# B&R Automation Studio project PLC code - cp (part 19)

#### InputsMecano.st - PhysicalInputs
```iecst
ACTION InputsMecano:

	//////////
	//PRINTER
	//////////

	// Machine controlled by line. Always with consent
	gMachine.In.xConsentL1Ok := TRUE;
	gMachine.In.xConsentL2Ok := TRUE;

	//Digital Inputs
	gMachine.In.Buttons.xStart := X20DIF371_101.DInput[1];
	gMachine.In.Buttons.xStop := NOT X20DIF371_101.DInput[2];
	gMachine.In.Buttons.xAuto := X20DIF371_101.DInput[3];
	gMachine.In.Buttons.xZero := NOT X20DIF371_101.DInput[4];
	gMachine.In.Buttons.xManual := X20DIF371_101.DInput[5];
	gMachine.In.Buttons.xReset := X20DIF371_101.DInput[6];
	//Back Safety Key unlock - PRINTER := X20DIF371_101.DInput[7];
	gBlockInputs[1].xReferenceDI := X20DIF371_101.DInput[8];
	gJamInputs[1].xJamLowCrash := X20DIF371_101.DInput[9];
	gJamInputs[2].xJamLowCrash := X20DIF371_101.DInput[10];
	gJamInputs[3].xJamLowCrash := X20DIF371_101.DInput[11];
	gJamInputs[1].xJamTestOk := X20DIF371_101.DInput[13];
	gJamInputs[2].xJamTestOk := X20DIF371_101.DInput[14];
	gJamInputs[3].xJamTestOk := X20DIF371_101.DInput[15];

	gBlockInputs[1].xPrintHeadPSU[1] := X20DIF371_102.DInput[1];
	gBlockInputs[1].xPrintHeadPSU[2] := X20DIF371_102.DInput[2];
	gBlockInputs[1].xPrintHeadPSU[3] := X20DIF371_102.DInput[3];
	gBlockInputs[1].xHeaterDcOkPsu[1] := gBlockInputs[1].xHeaterAcOkPsu[1] := X20DIF371_102.DInput[4];
	gInksInputs[3].xPrintHeadsPsuOK := X20DIF371_102.DInput[5];
	gInksInputs[4].xPrintHeadsPsuOK := X20DIF371_102.DInput[6];
	gInksInputs[5].xPrintHeadsPsuOK := X20DIF371_102.DInput[7];
	gInksInputs[6].xPrintHeadsPsuOK := X20DIF371_102.DInput[8];
	gInksInputs[7].xPrintHeadsPsuOK := X20DIF371_102.DInput[9];
	gInksInputs[8].xPrintHeadsPsuOK := X20DIF371_102.DInput[10];
	gInksInputs[9].xPrintHeadsPsuOK := X20DIF371_102.DInput[11];
	gInksInputs[10].xPrintHeadsPsuOK := X20DIF371_102.DInput[12];
	gMachine.In.x24Vdc := X20DIF371_102.DInput[13];
	gBelt.parameters.xDriveProtectionOK := X20DIF371_102.DInput[14];
	gBlockInputs[1].xDriveProtectionOK := gBlockInputs[1].xDifferentialOK := X20DIF371_102.DInput[15];
	FOR iIndexCuringLed:=1 TO MAX_LAST_CURING_LED DO
		gCuringLed[iIndexCuringLed].Signals.Inputs.xFrontDoorClosed := X20DIF371_102.DInput[16];
	END_FOR

	gMachine.In.ProductDetect.pPDSignalSensorL1	:= ADR(X20DIF371_103.DInput[1]);
	gMachine.In.ProductDetect.pPDSignalSensorL2	:= ADR(X20DIF371_103.DInput[2]);
	gPhotoCells.Inputs.Signals.pInput[1] := ADR(X20DIF371_103.DInput[3]);
	gPhotoCells.Inputs.Signals.pInput[2] := ADR(X20DIF371_103.DInput[4]);
	gPhotoCells.Inputs.Signals.pInput[3] := ADR(X20DIF371_103.DInput[5]);
	gPhotoCells.Inputs.Signals.pInput[4] := ADR(X20DIF371_103.DInput[6]);
	gPhotoCells.Inputs.Signals.pInput[5] := ADR(X20DIF371_103.DInput[7]);
	gPhotoCells.Inputs.Signals.pInput[6] := ADR(X20DIF371_103.DInput[8]);
	gPhotoCells.Inputs.Signals.xSafetyEnable := gMachine.In.xSafetyEnabled;

	gJamInputs[1].xJamCrash[1] := X20DIF371_104.DInput[1];
	gJamInputs[1].xJamCrash[2] := X20DIF371_104.DInput[2];
	gJamInputs[1].xJamCrash[3] := X20DIF371_104.DInput[3];
	gJamInputs[1].xJamCrash[4] := X20DIF371_104.DInput[4];
	gJamInputs[2].xJamCrash[1] := X20DIF371_104.DInput[5];
	gJamInputs[2].xJamCrash[2] := X20DIF371_104.DInput[6];
	gJamInputs[2].xJamCrash[3] := X20DIF371_104.DInput[7];
	gJamInputs[2].xJamCrash[4] := X20DIF371_104.DInput[8];
	gJamInputs[3].xJamCrash[1] := X20DIF371_104.DInput[9];
	gJamInputs[3].xJamCrash[2] := X20DIF371_104.DInput[10];

	gInksInputs[3].xKlixonTriggered := X20DIF371_105.DInput[1];
	gInksInputs[4].xKlixonTriggered := X20DIF371_105.DInput[2];
	gInksInputs[5].xKlixonTriggered := X20DIF371_105.DInput[3];
	gInksInputs[6].xKlixonTriggered := X20DIF371_105.DInput[4];
	gInksInputs[7].xKlixonTriggered := X20DIF371_105.DInput[5];
	gInksInputs[8].xKlixonTriggered := X20DIF371_105.DInput[6];
	gInksInputs[9].xKlixonTriggered := X20DIF371_105.DInput[7];
	gInksInputs[10].xKlixonTriggered := X20DIF371_105.DInput[8];

	gInksInputs[3].xOverpressure  := NOT X20DIF371_105.DInput[9];
	gInksInputs[4].xOverpressure  := NOT X20DIF371_105.DInput[10];
	gInksInputs[5].xOverpressure  := NOT X20DIF371_105.DInput[11];
	gInksInputs[6].xOverpressure  := NOT X20DIF371_105.DInput[12];
	gInksInputs[7].xOverpressure  := NOT X20DIF371_105.DInput[13];
	gInksInputs[8].xOverpressure  := NOT X20DIF371_105.DInput[14];
	gInksInputs[9].xOverpressure  := NOT X20DIF371_105.DInput[15];
	gInksInputs[10].xOverpressure  := NOT X20DIF371_105.DInput[16];

	gInksInputs[3].xConnected := X20DIF371_106.DInput[1];
	gInksInputs[4].xConnected := X20DIF371_106.DInput[2];
	gInksInputs[5].xConnected := X20DIF371_106.DInput[3];
	gInksInputs[6].xConnected := X20DIF371_106.DInput[4];
	gInksInputs[7].xConnected := X20DIF371_106.DInput[5];
	gInksInputs[8].xConnected := X20DIF371_106.DInput[6];
	gInksInputs[9].xConnected := X20DIF371_106.DInput[7];
	gInksInputs[10].xConnected := X20DIF371_106.DInput[8];

	//Analog inputs
	gTransVacuum[1].Inputs.iPressureRaw := X20AI8321_111.AInput[1];
	gTransVacuum[1].Inputs.xPressureSensorError := StatusAnalogInputBroken( X20AI8321_111.ModuleOk, X20AI8321_111.Status01, X20AI8321_111.Status02, 1);
	gTransVacuum[2].Inputs.iPressureRaw := X20AI8321_111.AInput[2];
	gTransVacuum[2].Inputs.xPressureSensorError := StatusAnalogInputBroken( X20AI8321_111.ModuleOk, X20AI8321_111.Status01, X20AI8321_111.Status02, 2);

	gInksInputs[3].iVacuum1Raw := X20AI8321_112.AInput[1];
	gInksInputs[3].xVacuum1SensorError 	:= StatusAnalogInputBroken( X20AI8321_112.ModuleOk, X20AI8321_112.Status01, X20AI8321_112.Status02, 1);
	gInksInputs[3].iVacuum2Raw := X20AI8321_112.AInput[2];
	gInksInputs[3].xVacuum2SensorError 	:= StatusAnalogInputBroken( X20AI8321_112.ModuleOk, X20AI8321_112.Status01, X20AI8321_112.Status02, 2);
	gInksInputs[4].iVacuum1Raw := X20AI8321_112.AInput[3];
	gInksInputs[4].xVacuum1SensorError 	:= StatusAnalogInputBroken( X20AI8321_112.ModuleOk, X20AI8321_112.Status01, X20AI8321_112.Status02, 3);
	gInksInputs[4].iVacuum2Raw := X20AI8321_112.AInput[4];
	gInksInputs[4].xVacuum2SensorError 	:= StatusAnalogInputBroken( X20AI8321_112.ModuleOk, X20AI8321_112.Status01, X20AI8321_112.Status02, 4);
	gInksInputs[5].iVacuum1Raw := X20AI8321_112.AInput[5];
	gInksInputs[5].xVacuum1SensorError 	:= StatusAnalogInputBroken( X20AI8321_112.ModuleOk, X20AI8321_112.Status01, X20AI8321_112.Status02, 5);
	gInksInputs[5].iVacuum2Raw := X20AI8321_112.AInput[6];
	gInksInputs[5].xVacuum2SensorError 	:= StatusAnalogInputBroken( X20AI8321_112.ModuleOk, X20AI8321_112.Status01, X20AI8321_112.Status02, 6);
	gInksInputs[6].iVacuum1Raw := X20AI8321_112.AInput[7];
	gInksInputs[6].xVacuum1SensorError 	:= StatusAnalogInputBroken( X20AI8321_112.ModuleOk, X20AI8321_112.Status01, X20AI8321_112.Status02, 7);
	gInksInputs[6].iVacuum2Raw := X20AI8321_112.AInput[8];
	gInksInputs[6].xVacuum2SensorError 	:= StatusAnalogInputBroken( X20AI8321_112.ModuleOk, X20AI8321_112.Status01, X20AI8321_112.Status02, 8);

	gInksInputs[7].iVacuum1Raw := X20AI8321_113.AInput[1];
	gInksInputs[7].xVacuum1SensorError 	:= StatusAnalogInputBroken( X20AI8321_113.ModuleOk, X20AI8321_113.Status01, X20AI8321_113.Status02, 1);
	gInksInputs[7].iVacuum2Raw := X20AI8321_113.AInput[2];
	gInksInputs[7].xVacuum2SensorError 	:= StatusAnalogInputBroken( X20AI8321_113.ModuleOk, X20AI8321_113.Status01, X20AI8321_113.Status02, 2);
	gInksInputs[8].iVacuum1Raw := X20AI8321_113.AInput[3];
	gInksInputs[8].xVacuum1SensorError 	:= StatusAnalogInputBroken( X20AI8321_113.ModuleOk, X20AI8321_113.Status01, X20AI8321_113.Status02, 3);
	gInksInputs[8].iVacuum2Raw := X20AI8321_113.AInput[4];
	gInksInputs[8].xVacuum2SensorError 	:= StatusAnalogInputBroken( X20AI8321_113.ModuleOk, X20AI8321_113.Status01, X20AI8321_113.Status02, 4);
	gInksInputs[9].iVacuum1Raw := X20AI8321_113.AInput[5];
	gInksInputs[9].xVacuum1SensorError 	:= StatusAnalogInputBroken( X20AI8321_113.ModuleOk, X20AI8321_113.Status01, X20AI8321_113.Status02, 5);
	gInksInputs[9].iVacuum2Raw := X20AI8321_113.AInput[6];
	gInksInputs[9].xVacuum2SensorError 	:= StatusAnalogInputBroken( X20AI8321_113.ModuleOk, X20AI8321_113.Status01, X20AI8321_113.Status02, 6);
	gInksInputs[10].iVacuum1Raw := X20AI8321_113.AInput[7];
	gInksInputs[10].xVacuum1SensorError 	:= StatusAnalogInputBroken( X20AI8321_113.ModuleOk, X20AI8321_113.Status01, X20AI8321_113.Status02, 7);
	gInksInputs[10].iVacuum2Raw := X20AI8321_113.AInput[8];
	gInksInputs[10].xVacuum2SensorError 	:= StatusAnalogInputBroken( X20AI8321_113.ModuleOk, X20AI8321_113.Status01, X20AI8321_113.Status02, 8);

	gInksInputs[3].iInTankLevel := X20AI8321_114.AInput[1];
	gInksInputs[3].xInkLevelTankSensorError := StatusAnalogInputBroken( X20AI8321_114.ModuleOk, X20AI8321_114.Status01, X20AI8321_114.Status02, 1);
	gInksInputs[4].iInTankLevel := X20AI8321_114.AInput[2];
	gInksInputs[4].xInkLevelTankSensorError := StatusAnalogInputBroken( X20AI8321_114.ModuleOk, X20AI8321_114.Status01, X20AI8321_114.Status02, 2);
	gInksInputs[5].iInTankLevel := X20AI8321_114.AInput[3];
	gInksInputs[5].xInkLevelTankSensorError := StatusAnalogInputBroken( X20AI8321_114.ModuleOk, X20AI8321_114.Status01, X20AI8321_114.Status02, 3);
	gInksInputs[6].iInTankLevel := X20AI8321_114.AInput[4];
	gInksInputs[6].xInkLevelTankSensorError := StatusAnalogInputBroken( X20AI8321_114.ModuleOk, X20AI8321_114.Status01, X20AI8321_114.Status02, 4);
	gInksInputs[7].iInTankLevel := X20AI8321_114.AInput[5];
	gInksInputs[7].xInkLevelTankSensorError := StatusAnalogInputBroken( X20AI8321_114.ModuleOk, X20AI8321_114.Status01, X20AI8321_114.Status02, 5);
	gInksInputs[8].iInTankLevel := X20AI8321_114.AInput[6];
	gInksInputs[8].xInkLevelTankSensorError := StatusAnalogInputBroken( X20AI8321_114.ModuleOk, X20AI8321_114.Status01, X20AI8321_114.Status02, 6);
	gInksInputs[9].iInTankLevel := X20AI8321_114.AInput[7];
	gInksInputs[9].xInkLevelTankSensorError := StatusAnalogInputBroken( X20AI8321_114.ModuleOk, X20AI8321_114.Status01, X20AI8321_114.Status02, 7);
	gInksInputs[10].iInTankLevel := X20AI8321_114.AInput[8];
	gInksInputs[10].xInkLevelTankSensorError := StatusAnalogInputBroken( X20AI8321_114.ModuleOk, X20AI8321_114.Status01, X20AI8321_114.Status02, 8);

	//PT100
	gBlockInputs[1].xModuleTemp01Ok	:= X20AT4222_120.ModuleOk;
	gInksInputs[3].iTemperatureRaw := X20AT4222_120.TempInput[1];
	gInksInputs[3].xTempSensorError	:= StatusTemperatureInput(X20AT4222_120.Status01, 1);
	gInksInputs[4].iTemperatureRaw := X20AT4222_120.TempInput[2];
	gInksInputs[4].xTempSensorError	:= StatusTemperatureInput(X20AT4222_120.Status01, 2);
	gInksInputs[5].iTemperatureRaw := X20AT4222_120.TempInput[3];
	gInksInputs[5].xTempSensorError	:= StatusTemperatureInput(X20AT4222_120.Status01, 3);
	gInksInputs[6].iTemperatureRaw := X20AT4222_120.TempInput[4];
	gInksInputs[6].xTempSensorError	:= StatusTemperatureInput(X20AT4222_120.Status01, 4);

	gBlockInputs[1].xModuleTemp02Ok	:= X20AT4222_121.ModuleOk;
	gInksInputs[7].iTemperatureRaw := X20AT4222_121.TempInput[1];
	gInksInputs[7].xTempSensorError	:= StatusTemperatureInput(X20AT4222_121.Status01, 1);
	gInksInputs[8].iTemperatureRaw := X20AT4222_121.TempInput[2];
	gInksInputs[8].xTempSensorError	:= StatusTemperatureInput(X20AT4222_121.Status01, 2);
	gInksInputs[9].iTemperatureRaw := X20AT4222_121.TempInput[3];
	gInksInputs[9].xTempSensorError	:= StatusTemperatureInput(X20AT4222_121.Status01, 3);
	gInksInputs[10].iTemperatureRaw := X20AT4222_121.TempInput[4];
	gInksInputs[10].xTempSensorError	:= StatusTemperatureInput(X20AT4222_121.Status01, 4);

	// SI UNIT BK1
	gBlockInputs[1].xSiUnitModuleOk		:= SiUnitPwrLnkBK1.ModuleOk;
	gMachine.In.xAirSupply				:= SiUnitPwrLnkBK1.Input01_16.0;
	gBlockInputs[1].xAirVenturiOK		:= SiUnitPwrLnkBK1.Input01_16.1;
	gBlockInputs[1].xTrayOut			:= SiUnitPwrLnkBK1.Input01_16.2;
	gBlockInputs[1].xIclaSensor			:= SiUnitPwrLnkBK1.Input01_16.3;
	gTransVacuum[1].Inputs.xVaccAirFlow	:= gTransVacuum[2].Inputs.xVaccAirFlow := SiUnitPwrLnkBK1.Input01_16.4; //No estamos haciendo nada con esto en el package de TransVacuum!
	gTransVacuum[1].Inputs.xJointSystemPressure:= gTransVacuum[2].Inputs.xJointSystemPressure := SiUnitPwrLnkBK1.Input01_16.5;
	gMachine.In.CleanBelt.xLowPosition 	:= SiUnitPwrLnkBK1.Input01_16.6;
	gMachine.In.CleanBelt.xHighPosition := SiUnitPwrLnkBK1.Input01_16.7;
	gBlockInputs[1].xBarsIn := TRUE;
	gTransVacuum[1].Inputs.xSafetyEnable := gTransVacuum[2].Inputs.xSafetyEnable := gMachine.In.xSafetyEnabled;

	//Signals Forced by Configuration
	gBlockInputs[1].Safety.xFrontEStopOK := gSafetyController.Inputs.xPrinterFrontsideEstop;
	gBlockInputs[1].Safety.xRearEStopOK := gSafetyController.Inputs.xPrinterBacksideEstop;

	gBlockInputs[1].Safety.xFrontSafetyOK	:= gSafetyController.Inputs.xPrinterFrontsideEstop AND gSafetyController.Inputs.xPrinterLightCurtain;
	gBlockInputs[1].Safety.xRearSafetyOK	:= gSafetyController.Inputs.xPrinterBacksideEstop AND gSafetyController.Inputs.xPrinterDoorLock;
	gBlockInputs[1].Safety.xSafetyOK 		:= gMachine.In.xSafetyEnabled;

	//There are no specific enables for light curtains. So we mapp PrinterLightCurtain status to these inputs to acknowledge that curtain is crossed
	gBlockInputs[1].Safety.xCurtainEnable01 := gBlockInputs[1].Safety.xCurtainEnable02 := gSafetyController.Inputs.xPrinterLightCurtain;

	//Signals Forced by Configuration
	FOR iIndexVac := 1 TO MAX_LAST_TRANS_VACUUM DO gTransVacuum[iIndexVac].Inputs.xBlowersAnyCB := FALSE; END_FOR

	///////////////////////////
	//UV Curing leds related

	//Digital inputs
	gCuringLed[iIndexColorCuringLedBar].Lamp[1].Inputs.ThermalFault	:= NOT X20DIF371_151.DInput[1];
	gCuringLed[iIndexColorCuringLedBar].Lamp[1].Inputs.SLMFault		:= NOT X20DIF371_151.DInput[2];
	gCuringLed[iIndexColorCuringLedBar].Lamp[2].Inputs.ThermalFault	:= NOT X20DIF371_151.DInput[3];
	gCuringLed[iIndexColorCuringLedBar].Lamp[2].Inputs.SLMFault		:= NOT X20DIF371_151.DInput[4];
	gCuringLed[iIndexColorCuringLedBar].Lamp[3].Inputs.ThermalFault	:= NOT X20DIF371_151.DInput[5];
	gCuringLed[iIndexColorCuringLedBar].Lamp[3].Inputs.SLMFault		:= NOT X20DIF371_151.DInput[6];
	gCuringLed[iIndexColorCuringLedBar].Lamp[4].Inputs.ThermalFault	:= NOT X20DIF371_151.DInput[7];
	gCuringLed[iIndexColorCuringLedBar].Lamp[4].Inputs.SLMFault		:= NOT X20DIF371_151.DInput[8];
	gCuringLed[iIndexColorCuringLedBar].Lamp[5].Inputs.ThermalFault	:= NOT X20DIF371_151.DInput[9];
	gCuringLed[iIndexColorCuringLedBar].Lamp[5].Inputs.SLMFault		:= NOT X20DIF371_151.DInput[10];
	gCuringLed[iIndexColorCuringLedBar].Signals.Inputs.xN2HighFlow	:= NOT X20DIF371_151.DInput[13];
	gCuringLed[iIndexColorCuringLedBar].Signals.Inputs.xN2LowFlow	:= NOT X20DIF371_151.DInput[14];

	gCuringLed[iIndexWhiteCuringLedBar].Lamp[1].Inputs.ThermalFault	:= NOT X20DIF371_152.DInput[1];
	gCuringLed[iIndexWhiteCuringLedBar].Lamp[1].Inputs.SLMFault		:= NOT X20DIF371_152.DInput[2];
	gCuringLed[iIndexWhiteCuringLedBar].Lamp[2].Inputs.ThermalFault	:= NOT X20DIF371_152.DInput[3];
	gCuringLed[iIndexWhiteCuringLedBar].Lamp[2].Inputs.SLMFault		:= NOT X20DIF371_152.DInput[4];
	gCuringLed[iIndexWhiteCuringLedBar].Lamp[3].Inputs.ThermalFault	:= NOT X20DIF371_152.DInput[5];
	gCuringLed[iIndexWhiteCuringLedBar].Lamp[3].Inputs.SLMFault		:= NOT X20DIF371_152.DInput[6];
	gCuringLed[iIndexWhiteCuringLedBar].Lamp[4].Inputs.ThermalFault	:= NOT X20DIF371_152.DInput[7];
	gCuringLed[iIndexWhiteCuringLedBar].Lamp[4].Inputs.SLMFault		:= NOT X20DIF371_152.DInput[8];
	gCuringLed[iIndexWhiteCuringLedBar].Lamp[5].Inputs.ThermalFault	:= NOT X20DIF371_152.DInput[9];
	gCuringLed[iIndexWhiteCuringLedBar].Lamp[5].Inputs.SLMFault		:= NOT X20DIF371_152.DInput[10];
	gCuringLed[iIndexWhiteCuringLedBar].Signals.Inputs.xN2HighFlow	:= NOT X20DIF371_152.DInput[13];
	gCuringLed[iIndexWhiteCuringLedBar].Signals.Inputs.xN2LowFlow	:= NOT X20DIF371_152.DInput[14];

	gCuringLed[iIndexPrimerCuringLedBar].Lamp[1].Inputs.ThermalFault	:= NOT X20DIF371_153.DInput[1];
	gCuringLed[iIndexPrimerCuringLedBar].Lamp[1].Inputs.SLMFault		:= NOT X20DIF371_153.DInput[2];
	gCuringLed[iIndexPrimerCuringLedBar].Lamp[2].Inputs.ThermalFault	:= NOT X20DIF371_153.DInput[3];
	gCuringLed[iIndexPrimerCuringLedBar].Lamp[2].Inputs.SLMFault		:= NOT X20DIF371_153.DInput[4];
	gCuringLed[iIndexPrimerCuringLedBar].Lamp[3].Inputs.ThermalFault	:= NOT X20DIF371_153.DInput[5];
	gCuringLed[iIndexPrimerCuringLedBar].Lamp[3].Inputs.SLMFault		:= NOT X20DIF371_153.DInput[6];
	gCuringLed[iIndexPrimerCuringLedBar].Lamp[4].Inputs.ThermalFault	:= NOT X20DIF371_153.DInput[7];
	gCuringLed[iIndexPrimerCuringLedBar].Lamp[4].Inputs.SLMFault		:= NOT X20DIF371_153.DInput[8];
	gCuringLed[iIndexPrimerCuringLedBar].Lamp[5].Inputs.ThermalFault	:= NOT X20DIF371_153.DInput[9];
	gCuringLed[iIndexPrimerCuringLedBar].Lamp[5].Inputs.SLMFault		:= NOT X20DIF371_153.DInput[10];
	gCuringLed[iIndexPrimerCuringLedBar].Signals.Inputs.xN2HighFlow		:= NOT X20DIF371_153.DInput[13];
	gCuringLed[iIndexPrimerCuringLedBar].Signals.Inputs.xN2LowFlow		:= NOT X20DIF371_153.DInput[14];

	gMachine.In.CleanBelt.xError 						:= X20DIF371_154.DInput[1];
	gMachine.In.CleanBelt.xOpenGuide 					:= X20DIF371_154.DInput[2];
	gMachine.In.AntiStatic.xGenAlarm 					:= X20DIF371_154.DInput[3];
	gMachine.In.AntiStatic.xIonLevelAlarm				:= X20DIF371_154.DInput[4];

	//////////
	//PDC
	//////////
	//Line X20DIF371_002
	//These inputs are read in MachineConfigurator>InputsMachineModel
	//	:= Pdc_X20DIF371_002.DInput[1];
	//	:= Pdc_X20DIF371_002.DInput[2];
	//	:= Pdc_X20DIF371_002.DInput[3];
	//	:= Pdc_X20DIF371_002.DInput[4];
	//	:= Pdc_X20DIF371_002.DInput[5];
	//	:= Pdc_X20DIF371_002.DInput[6];
	gFeeder.Inputs.xNoPowered 					:= NOT Pdc_X20DIF371_002.DInput[7];
	gSarm.Inputs.xPowered						:= Pdc_X20DIF371_002.DInput[8];
	gPrimer.Inputs.xNoPowered 					:= NOT Pdc_X20DIF371_002.DInput[9];
	gLine.Inputs.xPrinterPowered				:= Pdc_X20DIF371_002.DInput[10];
	gOverVarnish.Inputs.xNoPowered  			:= NOT Pdc_X20DIF371_002.DInput[11];
	gStacker.Inputs.xNoPowered 					:= NOT Pdc_X20DIF371_002.DInput[12];
	gLine.Inputs.xOvervoltageProtectionOk 		:= NOT Pdc_X20DIF371_002.DInput[13]; //Inverse logic
	gMachine.In.xSafetyEnabled 					:= Pdc_X20DIF371_002.DInput[14];

	//Line X20DIF371_003
	gAxisInverter[1].ElecSignals.In.xBreakerOK 	:= Pdc_X20DIF371_003.DInput[1];
	gAxisInverter[2].ElecSignals.In.xBreakerOK 	:= Pdc_X20DIF371_003.DInput[2];
	gAxisInverter[3].ElecSignals.In.xBreakerOK 	:= Pdc_X20DIF371_003.DInput[3];
	gAxisInverter[4].ElecSignals.In.xBreakerOK 	:= Pdc_X20DIF371_003.DInput[4];
	gMachine.In.xHoppersSoftStarterFault	:= Pdc_X20DIF371_003.DInput[5];
	gLine.Inputs.UPSs[1].LoadOnUtility		:= Pdc_X20DIF371_003.DInput[6];
	gLine.Inputs.UPSs[1].LoadOnBattery 		:= gLine.Inputs.UPSs[1].xPowerFault := Pdc_X20DIF371_003.DInput[7];
	gLine.Inputs.UPSs[1].xLowBattery 		:= Pdc_X20DIF371_003.DInput[8];
	gLine.Inputs.UPSs[1].xByPass			:= Pdc_X20DIF371_003.DInput[9];
	gLine.Inputs.x24VdcStartSeqNoPowered	:= NOT Pdc_X20DIF371_003.DInput[10];

	//Line X20DIF371_004
	gFeeder.Inputs.xModelInput[0] 		:= Pdc_X20DIF371_004.DInput[1];
	gFeeder.Inputs.xModelInput[1] 		:= Pdc_X20DIF371_004.DInput[2];
	gFeeder.Inputs.xModelInput[2] 		:= Pdc_X20DIF371_004.DInput[3];
	gFeeder.Inputs.xOnline 				:= Pdc_X20DIF371_004.DInput[4];
	gFeeder.Inputs.xError 				:= Pdc_X20DIF371_004.DInput[5];
	gFeeder.Inputs.xFeeding 			:= Pdc_X20DIF371_004.DInput[6];
	gFeeder.Inputs.xMultiPick 			:= Pdc_X20DIF371_004.DInput[7];
	gFeeder.Inputs.xTrayEmpty 			:= Pdc_X20DIF371_004.DInput[8];
	gFeeder.Inputs.xMediaLowL1 			:= Pdc_X20DIF371_004.DInput[9];
	gFeeder.Inputs.xMediaThickness 		:= Pdc_X20DIF371_004.DInput[10];
	gFeeder.Inputs.xReadyToFeed 		:= Pdc_X20DIF371_004.DInput[11];
	gSarm.Inputs.xModelInput[0] 		:= Pdc_X20DIF371_050.DInput[12];
	gSarm.Inputs.xModelInput[1] 		:= Pdc_X20DIF371_050.DInput[13];
	gSarm.Inputs.xModelInput[2] 		:= Pdc_X20DIF371_050.DInput[14];
	gSarm.Inputs.xError 				:= Pdc_X20DIF371_050.DInput[15];
	gSarm.Inputs.xRunning 				:= Pdc_X20DIF371_050.DInput[16];

	//Line X20DIF371_005
	gPrimer.Inputs.xModelInput[0] 		:= Pdc_X20DIF371_005.DInput[1];
	gPrimer.Inputs.xModelInput[1] 		:= Pdc_X20DIF371_005.DInput[2];
	gPrimer.Inputs.xModelInput[2] 		:= Pdc_X20DIF371_005.DInput[3];
	gPrimer.Inputs.xReadyToPrime 		:= Pdc_X20DIF371_004.DInput[4];
	gPrimer.Inputs.xCoating 			:= Pdc_X20DIF371_004.DInput[5];
	gPrimer.Inputs.xError 				:= Pdc_X20DIF371_004.DInput[6];
	gPrimer.Inputs.xDryerInRun 			:= Pdc_X20DIF371_005.DInput[7];
	gPrimer.Inputs.xTransportMoving 	:= Pdc_X20DIF371_005.DInput[8];
	gOverVarnish.Inputs.xModelInput[0] 	:= Pdc_X20DIF371_005.DInput[9];
	gOverVarnish.Inputs.xModelInput[1] 	:= Pdc_X20DIF371_005.DInput[10];
	gOverVarnish.Inputs.xModelInput[2] 	:= Pdc_X20DIF371_005.DInput[11];
	gOverVarnish.Inputs.xReadyToPrime 	:= Pdc_X20DIF371_005.DInput[12];
	gOverVarnish.Inputs.xCoating 		:= Pdc_X20DIF371_005.DInput[13];
	gOverVarnish.Inputs.xError 			:= Pdc_X20DIF371_005.DInput[14];
	gOverVarnish.Inputs.xDryerInRun 	:= Pdc_X20DIF371_005.DInput[15];
	gOverVarnish.Inputs.xTransportMoving := Pdc_X20DIF371_005.DInput[16];

	//Line X20DIF371_006
	gStacker.Inputs.xModelInput[0] 		:= Pdc_X20DIF371_006.DInput[1];
	gStacker.Inputs.xModelInput[1] 		:= Pdc_X20DIF371_006.DInput[2];
	gStacker.Inputs.xModelInput[2] 		:= Pdc_X20DIF371_006.DInput[3];
	gStacker.Inputs.xError 				:= Pdc_X20DIF371_006.DInput[4];
	gStacker.Inputs.xReadyToStack 		:= Pdc_X20DIF371_006.DInput[5];
	gStacker.Inputs.xFeedInterrupt 		:= Pdc_X20DIF371_006.DInput[6];
	gStacker.Inputs.xRunning 			:= Pdc_X20DIF371_006.DInput[7];
	gStacker.Inputs.xRejectSuccess 		:= Pdc_X20DIF371_006.DInput[8]; //En la excel de señales lo tienen al revés (aparece stacksucces), pero es porque creo que lo tienen mal en el cableado, así está bien.
	gStacker.Inputs.xStackSuccess 		:= Pdc_X20DIF371_006.DInput[9]; //En la excel de señales lo tienen al revés (aparece rejectsucces), pero es porque creo que lo tienen mal en el cableado, así está bien.

	//Line X20DIF371_020
	gCuringLed[iIndexColorCuringLedBar].Signals.Inputs.xPsuDcOk[1] := Pdc_X20DIF371_021.DInput[1];
	gCuringLed[iIndexColorCuringLedBar].Signals.Inputs.xPsuDcOk[2] := Pdc_X20DIF371_021.DInput[2];
	gCuringLed[iIndexColorCuringLedBar].Signals.Inputs.xPsuDcOk[3] := Pdc_X20DIF371_021.DInput[3];
	gCuringLed[iIndexColorCuringLedBar].Signals.Inputs.xPsuDcOk[4] := Pdc_X20DIF371_021.DInput[4];
	gCuringLed[iIndexColorCuringLedBar].Signals.Inputs.xPsuDcOk[5] := Pdc_X20DIF371_021.DInput[5];
	gCuringLed[iIndexColorCuringLedBar].Signals.Inputs.xPsuDcOk[6] := Pdc_X20DIF371_021.DInput[6];
	gCuringLed[iIndexColorCuringLedBar].Signals.Inputs.xPsuDcOk[7] := Pdc_X20DIF371_021.DInput[7];
	gCuringLed[iIndexColorCuringLedBar].Signals.Inputs.xPsuAcOk[1] := Pdc_X20DIF371_021.DInput[8];
	gCuringLed[iIndexColorCuringLedBar].Signals.Inputs.xPsuAcOk[2] := Pdc_X20DIF371_021.DInput[9];
	gCuringLed[iIndexColorCuringLedBar].Signals.Inputs.xPsuAcOk[3] := Pdc_X20DIF371_021.DInput[10];
	gCuringLed[iIndexColorCuringLedBar].Signals.Inputs.xPsuAcOk[4] := Pdc_X20DIF371_021.DInput[11];
	gCuringLed[iIndexColorCuringLedBar].Signals.Inputs.xPsuAcOk[5] := Pdc_X20DIF371_021.DInput[12];
	gCuringLed[iIndexColorCuringLedBar].Signals.Inputs.xPsuAcOk[6] := Pdc_X20DIF371_021.DInput[13];
	gCuringLed[iIndexColorCuringLedBar].Signals.Inputs.xPsuAcOk[7] := Pdc_X20DIF371_021.DInput[14];
	gCuringLed[iIndexColorCuringLedBar].Signals.Inputs.xSafetyEnable := gMachine.In.xSafetyEnabled;

	//Line X20DIF371_021
	gCuringLed[iIndexWhiteCuringLedBar].Signals.Inputs.xPsuDcOk[1] := Pdc_X20DIF371_022.DInput[1];
	gCuringLed[iIndexWhiteCuringLedBar].Signals.Inputs.xPsuDcOk[2] := Pdc_X20DIF371_022.DInput[2];
	gCuringLed[iIndexWhiteCuringLedBar].Signals.Inputs.xPsuDcOk[3] := Pdc_X20DIF371_022.DInput[3];
	gCuringLed[iIndexWhiteCuringLedBar].Signals.Inputs.xPsuDcOk[4] := Pdc_X20DIF371_022.DInput[4];
	gCuringLed[iIndexWhiteCuringLedBar].Signals.Inputs.xPsuDcOk[5] := Pdc_X20DIF371_022.DInput[5];
	gCuringLed[iIndexWhiteCuringLedBar].Signals.Inputs.xPsuDcOk[6] := Pdc_X20DIF371_022.DInput[6];
	gCuringLed[iIndexWhiteCuringLedBar].Signals.Inputs.xPsuDcOk[7] := Pdc_X20DIF371_022.DInput[7];
	gCuringLed[iIndexWhiteCuringLedBar].Signals.Inputs.xPsuAcOk[1] := Pdc_X20DIF371_022.DInput[8];
	gCuringLed[iIndexWhiteCuringLedBar].Signals.Inputs.xPsuAcOk[2] := Pdc_X20DIF371_022.DInput[9];
	gCuringLed[iIndexWhiteCuringLedBar].Signals.Inputs.xPsuAcOk[3] := Pdc_X20DIF371_022.DInput[10];
	gCuringLed[iIndexWhiteCuringLedBar].Signals.Inputs.xPsuAcOk[4] := Pdc_X20DIF371_022.DInput[11];
	gCuringLed[iIndexWhiteCuringLedBar].Signals.Inputs.xPsuAcOk[5] := Pdc_X20DIF371_022.DInput[12];
	gCuringLed[iIndexWhiteCuringLedBar].Signals.Inputs.xPsuAcOk[6] := Pdc_X20DIF371_022.DInput[13];
	gCuringLed[iIndexWhiteCuringLedBar].Signals.Inputs.xPsuAcOk[7] := Pdc_X20DIF371_022.DInput[14];
	gCuringLed[iIndexWhiteCuringLedBar].Signals.Inputs.xSafetyEnable := gMachine.In.xSafetyEnabled;

	//Line X20DIF371_023
	gCuringLed[iIndexPrimerCuringLedBar].Signals.Inputs.xPsuDcOk[1] := Pdc_X20DIF371_023.DInput[1];
	gCuringLed[iIndexPrimerCuringLedBar].Signals.Inputs.xPsuDcOk[2] := Pdc_X20DIF371_023.DInput[2];
	gCuringLed[iIndexPrimerCuringLedBar].Signals.Inputs.xPsuDcOk[3] := Pdc_X20DIF371_023.DInput[3];
	gCuringLed[iIndexPrimerCuringLedBar].Signals.Inputs.xPsuDcOk[4] := Pdc_X20DIF371_023.DInput[4];
	gCuringLed[iIndexPrimerCuringLedBar].Signals.Inputs.xPsuDcOk[5] := Pdc_X20DIF371_023.DInput[5];
	gCuringLed[iIndexPrimerCuringLedBar].Signals.Inputs.xPsuDcOk[6] := Pdc_X20DIF371_023.DInput[6];
	gCuringLed[iIndexPrimerCuringLedBar].Signals.Inputs.xPsuDcOk[7] := Pdc_X20DIF371_023.DInput[7];
	gCuringLed[iIndexPrimerCuringLedBar].Signals.Inputs.xPsuAcOk[1] := Pdc_X20DIF371_023.DInput[8];
	gCuringLed[iIndexPrimerCuringLedBar].Signals.Inputs.xPsuAcOk[2] := Pdc_X20DIF371_023.DInput[9];
	gCuringLed[iIndexPrimerCuringLedBar].Signals.Inputs.xPsuAcOk[3] := Pdc_X20DIF371_023.DInput[10];
	gCuringLed[iIndexPrimerCuringLedBar].Signals.Inputs.xPsuAcOk[4] := Pdc_X20DIF371_023.DInput[11];
	gCuringLed[iIndexPrimerCuringLedBar].Signals.Inputs.xPsuAcOk[5] := Pdc_X20DIF371_023.DInput[12];
	gCuringLed[iIndexPrimerCuringLedBar].Signals.Inputs.xPsuAcOk[6] := Pdc_X20DIF371_023.DInput[13];
	gCuringLed[iIndexPrimerCuringLedBar].Signals.Inputs.xPsuAcOk[7] := Pdc_X20DIF371_023.DInput[14];
	gCuringLed[iIndexPrimerCuringLedBar].Signals.Inputs.xSafetyEnable := gMachine.In.xSafetyEnabled;

	//Pdc_X20DIF371_023
	gChiller[gCuringLed[iIndexColorCuringLedBar].Parameters.iChillerIndex].In.xAlarm := Pdc_X20DIF371_024.DInput[1];
	gChiller[iIndexColorCuringLedBar].In.xCooling := Pdc_X20DIF371_024.DInput[2];
	gChiller[gCuringLed[iIndexWhiteCuringLedBar].Parameters.iChillerIndex].In.xAlarm := gChiller[gCuringLed[iIndexPrimerCuringLedBar].Parameters.iChillerIndex].In.xAlarm := Pdc_X20DIF371_024.DInput[3];
	gChiller[iIndexWhiteCuringLedBar].In.xCooling := gChiller[iIndexPrimerCuringLedBar].In.xCooling := Pdc_X20DIF371_024.DInput[4];

	//Signals Forced by Configuration
	FOR iIndexBlock := 1 TO gMachine.Pt.CT.iNumBlocks DO
		gBlockInputs[iIndexBlock].xHeaterDcOkBusBar1 := TRUE;
		gBlockInputs[iIndexBlock].xHeaterDcOkBusBar2 := TRUE;
		gBlock[iIndexBlock].parameters.Hw.iNumPrintheadsPSU := 3;
		gBlock[iIndexBlock].parameters.Hw.iNumHeaterPSU := 1;
	END_FOR

	//To review with electrical team how to get these signals from chiller
	gChiller[1].In.xPowered	:= TRUE;
	gChiller[2].In.xPowered	:= TRUE;

END_ACTION
```

### Program Logical/Printer/PhysicalMapping/PhysicalMapOutputs (IEC)

#### MappingOutputs.st - PhysicalInputs
```iecst
PROGRAM _CYCLIC

	//If in automation runtime, do not assign physical mapping
	IF gMachine.St.HwData.Family = FAMILY_BRAUTOMATIONRUNTIME THEN
		RETURN;
	END_IF

	CASE gMachine.Pt.MachineModel OF
		Type_P4_12B,
		Type_P4_12B_L,
		Type_P4_6B,
		Type_P4_CBK,
		Type_P4_6B_L:
			OutputsP4;

		Type_SHLD,
		Type_SHLD_L:
			OutputsShield;

		Type_S1400,
		Type_S1400_VAC_PWRLNK,
		Type_S1400_VAC_CAN:
			OutputsS1400;

		Type_P5_OIL,
		Type_P5_WTR:
			OutputsP5;

		Type_NOZ_2_AQ,
		Type_NOZ_2_UV,
		Type_NOZ_2_UV_White:
			OutputsNozomi2;

		Type_CUBE,
		Type_CUBE_INSPECTION,
		Type_CUBE_GULLIVER,
		Type_CUBE_GULLIVER_INSPECTION:
			OutputsCube;

		Type_MECANO_UV_WHITE,
		Type_MECANO_UV_OPV,
		Type_MECANO_UV_WHITE_OPV:
			OutputsMecano;

	END_CASE

END_PROGRAM
```

#### OutputsP4.st - PhysicalOutputs
```iecst
ACTION OutputsP4:

(*CABINET 01*)
	// X3 PLC
	X3.DOutput[1]:= gMachine.Out.xAirSupply;
	X3.DOutput[2]:= FALSE;
	X3.DOutput[3]:= FALSE;
	X3.DOutput[4]:= FALSE;

	X3.DOutput[8]:= FALSE;
	X3.DOutput[9]:= FALSE;
	X3.DOutput[10]:= FALSE;
	X3.DOutput[11]:= FALSE;
	X3.DOutput[12]:= FALSE;

	// X20DOF322_001
	X20DOF322_001.DOutput[1]:= gMachine.Out.xPC1Start;
	X20DOF322_001.DOutput[2]:= gMachine.Out.xPC2Start;
	X20DOF322_001.DOutput[3]:= gMachine.Out.xGreenLight;
	X20DOF322_001.DOutput[4]:= gMachine.Out.xBuzzerButtonPanel;
	X20DOF322_001.DOutput[5]:= gMachine.Out.xResetRouter;
	X20DOF322_001.DOutput[6]:= gMachine.Out.xResetCB1;
	X20DOF322_001.DOutput[7]:= gMachine.Out.xResetCB2;
	X20DOF322_001.DOutput[8]:= gMachine.Out.xConsentL1;
	X20DOF322_001.DOutput[9]:= gMachine.Out.xConsentL2;
	X20DOF322_001.DOutput[10]:= gMachine.Out.xCompenserLine1;
	X20DOF322_001.DOutput[11]:= gMachine.Out.xCompenserLine2;
	X20DOF322_001.DOutput[12]:= gMachine.Out.xYellowLight;
	X20DOF322_001.DOutput[13]:= gMachine.Out.xRedLight;
	X20DOF322_001.DOutput[14]:= gMachine.Out.xLine1ReadyToClean;
	X20DOF322_001.DOutput[15]:= gMachine.Out.xLine2ReadyToClean;
	X20DOF322_001.DOutput[16]:= gMachine.Out.xSuctionTurbine;

	// X20DOF322_004
	X20DOF322_004.DOutput[1]:= gMachine.Out.xLightReset;
	X20DOF322_004.DOutput[2]:= FALSE;
	X20DOF322_004.DOutput[3]:= FALSE;
	X20DOF322_004.DOutput[4]:= FALSE;
	X20DOF322_004.DOutput[5]:= FALSE;
	X20DOF322_004.DOutput[6]:= FALSE;
	X20DOF322_004.DOutput[7]:= FALSE;
	X20DOF322_004.DOutput[8]:= FALSE;
	X20DOF322_004.DOutput[9]:= FALSE;
	X20DOF322_004.DOutput[10]:= FALSE;
	X20DOF322_004.DOutput[11]:= FALSE;
	X20DOF322_004.DOutput[12]:= FALSE;
	X20DOF322_004.DOutput[13]:= FALSE;
	//02-23-2018 changed these outputs a common, Electrical changes in common to work with it
	X20DOF322_004.DOutput[14]:= gBlockOutputs[1].xEnableDobleShot OR gBlockOutputs[2].xEnableDobleShot;
	X20DOF322_004.DOutput[15]:= gBlockOutputs[1].xShotLine1 OR gBlockOutputs[2].xShotLine1;
	X20DOF322_004.DOutput[16]:= gBlockOutputs[1].xShotLine2 OR gBlockOutputs[2].xShotLine2;

	// X20AI2636_005
	X20AI2636_005.DOutput[1] := gDing.Out.xReset;;  // Reset the target fault

	// X20SLX402_006
	// Enable safety transport
	X20SLX402_006.DOutput[1]:= (NOT gMachine.In.Buttons.xZero) OR (gMachine.St.Mode.xAuto OR gMachine.St.Mode.xManual);

	(*CABINET 02*)

	// X20DOF322_106	 PRINTHEAD  AND RESISTORS POWER from 1 to 6 bars
	X20DOF322_106.DOutput[1]:= gInksOutputs[6].xOutPowPrintHead;
	X20DOF322_106.DOutput[2]:= gInksOutputs[5].xOutPowPrintHead;
	X20DOF322_106.DOutput[3]:= gInksOutputs[4].xOutPowPrintHead;
	X20DOF322_106.DOutput[4]:= gInksOutputs[3].xOutPowPrintHead;
	X20DOF322_106.DOutput[5]:= gInksOutputs[2].xOutPowPrintHead;
	X20DOF322_106.DOutput[6]:= gInksOutputs[1].xOutPowPrintHead;
	X20DOF322_106.DOutput[7]:= gInksOutputs[6].xOutBarResistance;
	X20DOF322_106.DOutput[8]:= gInksOutputs[5].xOutBarResistance;
	X20DOF322_106.DOutput[9]:= gInksOutputs[4].xOutBarResistance;
	X20DOF322_106.DOutput[10]:= gInksOutputs[3].xOutBarResistance;
	X20DOF322_106.DOutput[11]:= gInksOutputs[2].xOutBarResistance;
	X20DOF322_106.DOutput[12]:= gInksOutputs[1].xOutBarResistance;
	X20DOF322_106.DOutput[13]:= gInksOutputs[6].xOutResistanceTank;
	X20DOF322_106.DOutput[14]:= gInksOutputs[5].xOutResistanceTank;
	X20DOF322_106.DOutput[15]:= gInksOutputs[4].xOutResistanceTank;
	X20DOF322_106.DOutput[16]:= FALSE;

	// X20DOF322_107 	xSolenoid1 and xSolenoid2 from 1 to 6 bars
	X20DOF322_107.DOutput[1]:=  gInksOutputs[6].xSolenoid1;
	X20DOF322_107.DOutput[2]:=  gInksOutputs[6].xSolenoid2;
	X20DOF322_107.DOutput[3]:=  gInksOutputs[5].xSolenoid1;
	X20DOF322_107.DOutput[4]:=  gInksOutputs[5].xSolenoid2;
	X20DOF322_107.DOutput[5]:=  gInksOutputs[4].xSolenoid1;
	X20DOF322_107.DOutput[6]:=  gInksOutputs[4].xSolenoid2;
	X20DOF322_107.DOutput[7]:=  gInksOutputs[3].xSolenoid1;
	X20DOF322_107.DOutput[8]:=  gInksOutputs[3].xSolenoid2;
	X20DOF322_107.DOutput[9]:=  gInksOutputs[2].xSolenoid1;
	X20DOF322_107.DOutput[10]:= gInksOutputs[2].xSolenoid2;
	X20DOF322_107.DOutput[11]:= gInksOutputs[1].xSolenoid1;
	X20DOF322_107.DOutput[12]:= gInksOutputs[1].xSolenoid2;
	X20DOF322_107.DOutput[13]:= gInksOutputs[3].xOutResistanceTank;
	X20DOF322_107.DOutput[14]:= gInksOutputs[2].xOutResistanceTank;
	X20DOF322_107.DOutput[15]:= gInksOutputs[1].xOutResistanceTank;
	X20DOF322_107.DOutput[16]:= FALSE;

	// X20DOF322_108						// Enable curtain is not connected here because was changed by EE team
	X20DOF322_108.DOutput[1]:= FALSE; 	//gBlockOutputs[1].xEnableCurtain;
	X20DOF322_108.DOutput[2]:= FALSE;
	X20DOF322_108.DOutput[3]:= gInksOutputs[6].xReliefValve; // SEIKO L relief valve BAR A
	X20DOF322_108.DOutput[4]:= gInksOutputs[5].xReliefValve; // SEIKO L relief valve BAR B XXXXXXXXXXXXXXXXXXXXXXXXX
	X20DOF322_108.DOutput[5]:= gInksOutputs[4].xReliefValve; // SEIKO L relief valve BAR C
	X20DOF322_108.DOutput[6]:= gInksOutputs[3].xReliefValve; // SEIKO L relief valve BAR D
	X20DOF322_108.DOutput[7]:= gInksOutputs[2].xReliefValve; // SEIKO L relief valve BAR E OOOOOOOOOOOOOOOOOOOOOOOOOO
	X20DOF322_108.DOutput[8]:= gInksOutputs[1].xReliefValve; // SEIKO L relief valve BAR F
	X20DOF322_108.DOutput[9]:= FALSE;
	X20DOF322_108.DOutput[10]:= FALSE;
	X20DOF322_108.DOutput[11]:= FALSE;
	X20DOF322_108.DOutput[12]:= FALSE;
	X20DOF322_108.DOutput[13]:= FALSE;
	//02-23-2018 changed these outputs a common, for that now are these outputs are always false in block
	//	X20DOF322_108.DOutput[14]:= gBlockOutputs[1].xShotLine1;
	//	X20DOF322_108.DOutput[15]:= gBlockOutputs[1].xShotLine2;
	//	X20DOF322_108.DOutput[16]:= gBlockOutputs[1].xEnableDobleShot;
	X20DOF322_108.DOutput[14]:= FALSE;
	X20DOF322_108.DOutput[15]:= FALSE;
	X20DOF322_108.DOutput[16]:= FALSE;

	// X20AO4622_111 	(*  BAR F *) 	(*  BAR E *)
	X20AO4622_111.AOutput[1]:= gInksOutputs[6].iDutyCycleNegative;
	X20AO4622_111.AOutput[2]:= gInksOutputs[6].iDutyCycleFilling;
	X20AO4622_111.AOutput[3]:= gInksOutputs[5].iDutyCycleNegative;
	X20AO4622_111.AOutput[4]:= gInksOutputs[5].iDutyCycleFilling;

	// X20AO4622_112	 (*  BAR D *)	 (*  BAR C *)
	X20AO4622_112.AOutput[1]:= gInksOutputs[4].iDutyCycleNegative;
	X20AO4622_112.AOutput[2]:= gInksOutputs[4].iDutyCycleFilling;
	X20AO4622_112.AOutput[3]:= gInksOutputs[3].iDutyCycleNegative;
	X20AO4622_112.AOutput[4]:= gInksOutputs[3].iDutyCycleFilling;

	// X20AO4622_113	 (*  BAR B *)	 (*  BAR A *)
	X20AO4622_113.AOutput[1]:= gInksOutputs[2].iDutyCycleNegative;
	X20AO4622_113.AOutput[2]:= gInksOutputs[2].iDutyCycleFilling;
	X20AO4622_113.AOutput[3]:= gInksOutputs[1].iDutyCycleNegative;
	X20AO4622_113.AOutput[4]:= gInksOutputs[1].iDutyCycleFilling;

	// X20SO2110_118
	X20SO2110_118.DOutput[1]:=gBlockOutputs[1].xEnableDrive;
	X20SO2110_118.DOutput[2]:=gBlockOutputs[1].xEnableIclaSI;

	// SI UNIT BK1
	SiUnitBK1.Output01_08.0	:= gBlockOutputs[1].xTrayIn;
	SiUnitBK1.Output01_08.1	:= gBlockOutputs[1].xTrayOut;
	SiUnitBK1.Output01_08.2	:= gMachine.commands.CleanBelt.xCleanBeltPump;
	SiUnitBK1.Output01_08.3	:= gBlockOutputs[1].xVenturi;
	SiUnitBK1.Output01_08.4	:= gMachine.commands.CleanBelt.xPistonFlojet;
	SiUnitBK1.Output01_08.5	:= gBlockOutputs[1].xCleaningWaterPump;

	(*CABINET 03*)

	// X20DOF322_206 PRINTHEAD  AND RESISTORS POWER from 7 to 12 bars
	X20DOF322_206.DOutput[1]:= gInksOutputs[12].xOutPowPrintHead;
	X20DOF322_206.DOutput[2]:= gInksOutputs[11].xOutPowPrintHead;
	X20DOF322_206.DOutput[3]:= gInksOutputs[10].xOutPowPrintHead;
	X20DOF322_206.DOutput[4]:= gInksOutputs[9].xOutPowPrintHead;
	X20DOF322_206.DOutput[5]:= gInksOutputs[8].xOutPowPrintHead;
	X20DOF322_206.DOutput[6]:= gInksOutputs[7].xOutPowPrintHead;
	X20DOF322_206.DOutput[7]:= gInksOutputs[12].xOutBarResistance;
	X20DOF322_206.DOutput[8]:= gInksOutputs[11].xOutBarResistance;
	X20DOF322_206.DOutput[9]:= gInksOutputs[10].xOutBarResistance;
	X20DOF322_206.DOutput[10]:= gInksOutputs[9].xOutBarResistance;
	X20DOF322_206.DOutput[11]:= gInksOutputs[8].xOutBarResistance;
	X20DOF322_206.DOutput[12]:= gInksOutputs[7].xOutBarResistance;
	X20DOF322_206.DOutput[13]:= gInksOutputs[12].xOutResistanceTank;
	X20DOF322_206.DOutput[14]:= gInksOutputs[11].xOutResistanceTank;
	X20DOF322_206.DOutput[15]:= gInksOutputs[10].xOutResistanceTank;
	X20DOF322_206.DOutput[16]:= FALSE;

	// X20DOF322_207
	X20DOF322_207.DOutput[1]:= gInksOutputs[12].xSolenoid1;
	X20DOF322_207.DOutput[2]:= gInksOutputs[12].xSolenoid2;
	X20DOF322_207.DOutput[3]:= gInksOutputs[11].xSolenoid1;
	X20DOF322_207.DOutput[4]:= gInksOutputs[11].xSolenoid2;
	X20DOF322_207.DOutput[5]:= gInksOutputs[10].xSolenoid1;
	X20DOF322_207.DOutput[6]:= gInksOutputs[10].xSolenoid2;
	X20DOF322_207.DOutput[7]:= gInksOutputs[9].xSolenoid1;
	X20DOF322_207.DOutput[8]:= gInksOutputs[9].xSolenoid2;
	X20DOF322_207.DOutput[9]:= gInksOutputs[8].xSolenoid1;
	X20DOF322_207.DOutput[10]:= gInksOutputs[8].xSolenoid2;
	X20DOF322_207.DOutput[11]:= gInksOutputs[7].xSolenoid1;
	X20DOF322_207.DOutput[12]:= gInksOutputs[7].xSolenoid2;
	X20DOF322_207.DOutput[13]:= gInksOutputs[9].xOutResistanceTank;
	X20DOF322_207.DOutput[14]:= gInksOutputs[8].xOutResistanceTank;
	X20DOF322_207.DOutput[15]:= gInksOutputs[7].xOutResistanceTank;
	X20DOF322_207.DOutput[16]:= FALSE;

	// X20DOF322_208						// Enable curtain is not connected here because was changed by EE team
	X20DOF322_208.DOutput[1]:= FALSE; 	//gBlockOutputs[2].xEnableCurtain;
	X20DOF322_208.DOutput[2]:= FALSE;
	X20DOF322_208.DOutput[3]:= gInksOutputs[12].xReliefValve; // SEIKO L relief valve BAR G
	X20DOF322_208.DOutput[4]:= gInksOutputs[11].xReliefValve; // SEIKO L relief valve BAR H
	X20DOF322_208.DOutput[5]:= gInksOutputs[10].xReliefValve; // SEIKO L relief valve BAR I
	X20DOF322_208.DOutput[6]:= gInksOutputs[9].xReliefValve;  // SEIKO L relief valve BAR K
	X20DOF322_208.DOutput[7]:= gInksOutputs[8].xReliefValve;  // SEIKO L relief valve BAR K
	X20DOF322_208.DOutput[8]:= gInksOutputs[7].xReliefValve;  // SEIKO L relief valve BAR L
	X20DOF322_208.DOutput[9]:= FALSE;
	X20DOF322_208.DOutput[10]:= FALSE;
	X20DOF322_208.DOutput[11]:= FALSE;
	X20DOF322_208.DOutput[12]:= FALSE;
	X20DOF322_208.DOutput[13]:= FALSE;
	//02-23-2018 changed these outputs a common, for that now are these outputs are always false in block
	//	X20DOF322_208.DOutput[14]:= gBlockOutputs[2].xShotLine1;
	//	X20DOF322_208.DOutput[15]:= gBlockOutputs[2].xShotLine2;
	//	X20DOF322_208.DOutput[16]:= gBlockOutputs[2].xEnableDobleShot;
	X20DOF322_208.DOutput[14]:= FALSE;
	X20DOF322_208.DOutput[15]:= FALSE;
	X20DOF322_208.DOutput[16]:= FALSE;

	// X20AO4622_211
	X20AO4622_211.AOutput[1] 	:= gInksOutputs[12].iDutyCycleNegative;
	X20AO4622_211.AOutput[2] 	:= gInksOutputs[12].iDutyCycleFilling;
	X20AO4622_211.AOutput[3] 	:= gInksOutputs[11].iDutyCycleNegative;
	X20AO4622_211.AOutput[4] 	:= gInksOutputs[11].iDutyCycleFilling;
	//BAR PUMP

	// X20AO4622_212
	X20AO4622_212.AOutput[1] 	:= gInksOutputs[10].iDutyCycleNegative;
	X20AO4622_212.AOutput[2] 	:= gInksOutputs[10].iDutyCycleFilling;
	X20AO4622_212.AOutput[3] 	:= gInksOutputs[9].iDutyCycleNegative;
	X20AO4622_212.AOutput[4] 	:= gInksOutputs[9].iDutyCycleFilling;

	// X20AO4622_213
	X20AO4622_213.AOutput[1] 	:= gInksOutputs[8].iDutyCycleNegative;
	X20AO4622_213.AOutput[2] 	:= gInksOutputs[8].iDutyCycleFilling;
	X20AO4622_213.AOutput[3] 	:= gInksOutputs[7].iDutyCycleNegative;
	X20AO4622_213.AOutput[4] 	:= gInksOutputs[7].iDutyCycleFilling;

	// X20SO2110_218
	X20SO2110_218.DOutput[1]:=gBlockOutputs[2].xEnableDrive;
	X20SO2110_218.DOutput[2]:=gBlockOutputs[2].xEnableIclaSI;

	// SI UNIT BK2
	SiUnitBK2.Output01_08.0:= gBlockOutputs[2].xTrayIn;
	SiUnitBK2.Output01_08.1:= gBlockOutputs[2].xTrayOut;
	SiUnitBK2.Output01_08.2:= gMachine.commands.CleanBelt.xCleanBeltPump;
	SiUnitBK2.Output01_08.3:= gBlockOutputs[2].xVenturi;
	SiUnitBK2.Output01_08.4:= gMachine.commands.CleanBelt.xPistonFlojet;
	SiUnitBK2.Output01_08.5	:= gBlockOutputs[2].xCleaningWaterPump;

END_ACTION
```

#### OutputsS1400.st - PhysicalOutputs
```iecst
ACTION OutputsS1400:

(*CABINET 01*)

	//X20DOF322_009
	X20DOF322_009.DOutput[1]:=gBlockOutputs[1].xShotLine1;
	X20DOF322_009.DOutput[2]:=gBlockOutputs[1].xShotLine2;
	X20DOF322_009.DOutput[3]:=gBlockOutputs[1].xEnableDobleShot;
	X20DOF322_009.DOutput[4]:=gMachine.Out.xResetCB1;
	X20DOF322_009.DOutput[5]:=gMachine.Out.xResetRouter;
	X20DOF322_009.DOutput[6]:= FALSE;								//SPARE
	X20DOF322_009.DOutput[7]:=gMachine.Out.xAirSupply;
	X20DOF322_009.DOutput[8]:=gMachine.Out.xGreenLight;
	X20DOF322_009.DOutput[9]:=gMachine.Out.xLightReset;
	X20DOF322_009.DOutput[10]:=gMachine.Out.xBuzzerButtonPanel;
	X20DOF322_009.DOutput[11]:= TRUE;
	X20DOF322_009.DOutput[12]:= FALSE;								//SPARE
	X20DOF322_009.DOutput[13]:= FALSE;								//SPARE
	X20DOF322_009.DOutput[14]:= FALSE;								//SPARE
	X20DOF322_009.DOutput[15]:= FALSE;								//SPARE
	X20DOF322_009.DOutput[16]:= FALSE;								//SPARE

	// X20DOF322_010
	X20DOF322_010.DOutput[1]:= gInksOutputs[1].xOutPowPrintHead;
	X20DOF322_010.DOutput[2]:= gInksOutputs[2].xOutPowPrintHead;
	X20DOF322_010.DOutput[3]:= gInksOutputs[3].xOutPowPrintHead;
	X20DOF322_010.DOutput[4]:= gInksOutputs[4].xOutPowPrintHead;
	X20DOF322_010.DOutput[5]:= gInksOutputs[5].xOutPowPrintHead;
	X20DOF322_010.DOutput[6]:= gInksOutputs[6].xOutPowPrintHead;
	X20DOF322_010.DOutput[7]:= gInksOutputs[7].xOutPowPrintHead;
	X20DOF322_010.DOutput[8]:= gInksOutputs[8].xOutPowPrintHead;
	X20DOF322_010.DOutput[9]:= gInksOutputs[1].xOutBarResistance;
	X20DOF322_010.DOutput[10]:= gInksOutputs[2].xOutBarResistance;
	X20DOF322_010.DOutput[11]:= gInksOutputs[3].xOutBarResistance;
	X20DOF322_010.DOutput[12]:= gInksOutputs[4].xOutBarResistance;
	X20DOF322_010.DOutput[13]:= gInksOutputs[5].xOutBarResistance;
	X20DOF322_010.DOutput[14]:= gInksOutputs[6].xOutBarResistance;
	X20DOF322_010.DOutput[15]:= gInksOutputs[7].xOutBarResistance;
	X20DOF322_010.DOutput[16]:= gInksOutputs[8].xOutBarResistance;

	//X20DOF322_011
	X20DOF322_011.DOutput[1] := gInksOutputs[1].xSolenoid1;
	X20DOF322_011.DOutput[2] := gInksOutputs[2].xSolenoid1;
	X20DOF322_011.DOutput[3] := gInksOutputs[1].xSolenoid2;
	X20DOF322_011.DOutput[4] := gInksOutputs[2].xSolenoid2;
	X20DOF322_011.DOutput[5] := gInksOutputs[3].xSolenoid1;
	X20DOF322_011.DOutput[6] := gInksOutputs[4].xSolenoid1;
	X20DOF322_011.DOutput[7] := gInksOutputs[3].xSolenoid2;
	X20DOF322_011.DOutput[8] := gInksOutputs[4].xSolenoid2;
	X20DOF322_011.DOutput[9] := gInksOutputs[5].xSolenoid1;
	X20DOF322_011.DOutput[10] := gInksOutputs[6].xSolenoid1;
	X20DOF322_011.DOutput[11] := gInksOutputs[5].xSolenoid2;
	X20DOF322_011.DOutput[12] := gInksOutputs[6].xSolenoid2;
	X20DOF322_011.DOutput[13] := gInksOutputs[7].xSolenoid1;
	X20DOF322_011.DOutput[14] := gInksOutputs[8].xSolenoid1;
	X20DOF322_011.DOutput[15] := gInksOutputs[7].xSolenoid2;
	X20DOF322_011.DOutput[16] := gInksOutputs[8].xSolenoid2;

	//X20DOF322_012
	X20DOF322_012.DOutput[1]:=gInksOutputs[1].xReliefValve;
	X20DOF322_012.DOutput[2]:=gInksOutputs[2].xReliefValve;
	X20DOF322_012.DOutput[3]:=gInksOutputs[3].xReliefValve;
	X20DOF322_012.DOutput[4]:=gInksOutputs[4].xReliefValve;
	X20DOF322_012.DOutput[5]:=gInksOutputs[5].xReliefValve;
	X20DOF322_012.DOutput[6]:=gInksOutputs[6].xReliefValve;
	X20DOF322_012.DOutput[7]:=gInksOutputs[7].xReliefValve;
	X20DOF322_012.DOutput[8]:=gInksOutputs[8].xReliefValve;
	X20DOF322_012.DOutput[9]:= FALSE;								//SPARE
	X20DOF322_012.DOutput[10]:=FALSE;								//SPARE
	X20DOF322_012.DOutput[11]:=FALSE;								//SPARE
	X20DOF322_012.DOutput[12]:=FALSE;								//SPARE
	X20DOF322_012.DOutput[13]:=FALSE;								//SPARE
	X20DOF322_012.DOutput[14]:=FALSE;								//SPARE
	X20DOF322_012.DOutput[15]:=FALSE;								//SPARE
	X20DOF322_012.DOutput[16]:=FALSE;								//SPARE

	//X20DOF322_013
	X20DOF322_013.DOutput[1]:=gMachine.Out.xConsentL1;
	X20DOF322_013.DOutput[2]:=gMachine.Out.xConsentL2;
	X20DOF322_013.DOutput[3]:=gMachine.Out.xCompenserLine1;
	X20DOF322_013.DOutput[4]:=gMachine.Out.xCompenserLine2;
	X20DOF322_013.DOutput[5]:=gMachine.Out.xYellowLight;
	X20DOF322_013.DOutput[6]:=gMachine.Out.xRedLight;
	X20DOF322_013.DOutput[7]:=gMachine.Out.xLine1ReadyToClean;
	X20DOF322_013.DOutput[8]:=gMachine.Out.xLine2ReadyToClean;
	X20DOF322_013.DOutput[9]:=gMachine.Out.xSuctionTurbine;
	X20DOF322_013.DOutput[10]:= gJamDetect[1].Outputs.xJamTestSignal[1] OR gJamDetect[2].Outputs.xJamTestSignal[1];
	X20DOF322_013.DOutput[11]:=gJamDetect[1].Outputs.xJamTestSignal[2] OR gJamDetect[2].Outputs.xJamTestSignal[2];
	X20DOF322_013.DOutput[12]:=gJamDetect[1].Outputs.xJamTestSignal[3] OR gJamDetect[2].Outputs.xJamTestSignal[3];
	X20DOF322_013.DOutput[13]:=gJamDetect[1].Outputs.xJamTestSignal[4] OR gJamDetect[2].Outputs.xJamTestSignal[4];
	X20DOF322_013.DOutput[14]:= FALSE;								//SPARE
	X20DOF322_013.DOutput[15]:= FALSE;								//SPARE
	X20DOF322_013.DOutput[16]:= FALSE;								//SPARE

	// X20AO4622_017 	(*  BAR A *) 	(*  BAR B *)
	X20AO4622_017.AOutput[1]:= gInksOutputs[1].iDutyCycleNegative;
	X20AO4622_017.AOutput[2]:= gInksOutputs[2].iDutyCycleNegative;
	X20AO4622_017.AOutput[3]:= gInksOutputs[1].iDutyCycleFilling;
	X20AO4622_017.AOutput[4]:= gInksOutputs[2].iDutyCycleFilling;

	// X20AO4622_018 	(*  BAR C *) 	(*  BAR D *)
	X20AO4622_018.AOutput[1]:= gInksOutputs[3].iDutyCycleNegative;
	X20AO4622_018.AOutput[2]:= gInksOutputs[4].iDutyCycleNegative;
	X20AO4622_018.AOutput[3]:= gInksOutputs[3].iDutyCycleFilling;
	X20AO4622_018.AOutput[4]:= gInksOutputs[4].iDutyCycleFilling;

	// X20AO4622_019 	(*  BAR E *) 	(*  BAR F *)
	X20AO4622_019.AOutput[1]:= gInksOutputs[5].iDutyCycleNegative;
	X20AO4622_019.AOutput[2]:= gInksOutputs[6].iDutyCycleNegative;
	X20AO4622_019.AOutput[3]:= gInksOutputs[5].iDutyCycleFilling;
	X20AO4622_019.AOutput[4]:= gInksOutputs[6].iDutyCycleFilling;

	// X20AO4622_020 	(*  BAR G *) 	(*  BAR H *)
	X20AO4622_020.AOutput[1]:= gInksOutputs[7].iDutyCycleNegative;
	X20AO4622_020.AOutput[2]:= gInksOutputs[8].iDutyCycleNegative;
	X20AO4622_020.AOutput[3]:= gInksOutputs[7].iDutyCycleFilling;
	X20AO4622_020.AOutput[4]:= gInksOutputs[8].iDutyCycleFilling;

	// X20AO4622_100 THICKNESS SENSOR RESET
	X20AI2636_100.DOutput[1] := gDing.Out.xReset;;  // Reset the target fault

	// SI UNIT BK1
	SiUnitPwrLnkBK1.Output01_16.0 := gBlockOutputs[1].xTrayIn;
	SiUnitPwrLnkBK1.Output01_16.1 := gBlockOutputs[1].xTrayOut;
	SiUnitPwrLnkBK1.Output01_16.2 := gMachine.commands.CleanBelt.xCleanBeltPump;
	SiUnitPwrLnkBK1.Output01_16.3 := gBlockOutputs[1].xVenturi;
	SiUnitPwrLnkBK1.Output01_16.4 := gBlockOutputs[1].xCleaningWaterPump;
	SiUnitPwrLnkBK1.Output01_16.5 := gMachine.commands.CleanBelt.xPistonFlojet;
	SiUnitPwrLnkBK1.Output01_16.6 := gMachine.commands.CleanBelt.xCleanBeltTopScraper;
	SiUnitPwrLnkBK1.Output01_16.7 := FALSE;

	//Vacuum
	SiUnitPwrLnkBK1.Output01_16.8 := gTransVacuum[1].Outputs.VacuumValves.0;
	SiUnitPwrLnkBK1.Output01_16.9 := gTransVacuum[1].Outputs.VacuumValves.1;
	SiUnitPwrLnkBK1.Output01_16.10 := gTransVacuum[1].Outputs.VacuumValves.2;
	SiUnitPwrLnkBK1.Output01_16.11 := gTransVacuum[1].Outputs.VacuumValves.3;
	SiUnitPwrLnkBK1.Output01_16.12 := gTransVacuum[1].Outputs.VacuumValves.4;
	SiUnitPwrLnkBK1.Output01_16.13 := gTransVacuum[1].Outputs.VacuumValves.5;
	SiUnitPwrLnkBK1.Output01_16.14 := gTransVacuum[1].Outputs.VacuumValves.6;
	SiUnitPwrLnkBK1.Output01_16.15 := gTransVacuum[1].Outputs.VacuumValves.7;
	SiUnitPwrLnkBK1.Output17_32.0 := gTransVacuum[1].Outputs.VacuumValves.8;
	SiUnitPwrLnkBK1.Output17_32.1 := gTransVacuum[1].Outputs.VacuumValves.9;
	SiUnitPwrLnkBK1.Output17_32.2 := gTransVacuum[1].Outputs.VacuumValves.10;
	SiUnitPwrLnkBK1.Output17_32.3 := gTransVacuum[1].Outputs.VacuumValves.11;
	SiUnitPwrLnkBK1.Output17_32.4 := gTransVacuum[1].Outputs.VacuumValves.12;
	SiUnitPwrLnkBK1.Output17_32.5 := gTransVacuum[1].Outputs.VacuumValves.13;
	SiUnitPwrLnkBK1.Output17_32.6 := gTransVacuum[1].Outputs.VacuumValves.14;
	SiUnitPwrLnkBK1.Output17_32.7 := gTransVacuum[1].Outputs.VacuumValves.15;
	SiUnitPwrLnkBK1.Output17_32.8 := gTransVacuum[1].Outputs.VacuumValves.16;
	SiUnitPwrLnkBK1.Output17_32.9 := gTransVacuum[1].Outputs.VacuumValves.17;
	SiUnitPwrLnkBK1.Output17_32.10 := gTransVacuum[1].Outputs.VacuumValves.18;
	SiUnitPwrLnkBK1.Output17_32.11 := gTransVacuum[1].Outputs.VacuumValves.19;

END_ACTION
```

#### OutputsCube.st - PhysicalOutputs
```iecst
ACTION OutputsCube:
	//////////
	//PDC
	//////////
	//KE008
	Pdc_X20DOF322_005.DOutput[1] := gMachine.In.xPowerSwitch; //Belt power circuit
	Pdc_X20DOF322_005.DOutput[2] := gMachine.In.xPowerSwitch; //Block power circuit
	Pdc_X20DOF322_005.DOutput[3] := gMachine.In.xPowerSwitch; //Fans activation
	Pdc_X20DOF322_005.DOutput[4] := gMachine.In.xPowerSwitch; //Control 24Vdc
	Pdc_X20DOF322_005.DOutput[5] := gMachine.In.xPowerSwitch; //IDS 24Vdc
	Pdc_X20DOF322_005.DOutput[6] := gMachine.In.xPowerSwitch; //Load 24Vdc
	Pdc_X20DOF322_005.DOutput[7] :=  gMachine.St.Remote.xSafetyReadyToReset;
	Pdc_X20DOF322_005.DOutput[8] :=  gMachine.St.Remote.xBeltNotStopped;
	Pdc_X20DOF322_005.DOutput[9] :=  gThicknessCtrl.Outputs.xReject;
	Pdc_X20DOF322_005.DOutput[10] := gThicknessCtrl.status.Reject.xRejecting;
	//Pdc_X20DOF322_005.DOutput[11] := ;
	//Pdc_X20DOF322_005.DOutput[12] := ;
	//Pdc_X20DOF322_005.DOutput[13] := ;
	//Pdc_X20DOF322_005.DOutput[14] := ;
	//Pdc_X20DOF322_005.DOutput[15] := ;
	//Pdc_X20DOF322_005.DOutput[16] := ;

	////KE010
	Pdc_X20DOF322_007.DOutput[1] := gMachine.Out.xResetHub;
	Pdc_X20DOF322_007.DOutput[2] := gMachine.Out.xResetSwitch;
	Pdc_X20DOF322_007.DOutput[3] := NOT gSafetyController.Inputs.xPrinterDoorLock; //Internal lights. ¿How shoud be controlled this?
	Pdc_X20DOF322_007.DOutput[4] := gMachine.Out.xWhiteLight;
	Pdc_X20DOF322_007.DOutput[5] := gMachine.Out.xRedLight;
	Pdc_X20DOF322_007.DOutput[6] := gMachine.Out.xGreenLight;
	Pdc_X20DOF322_007.DOutput[7] := gMachine.Out.xBlueLight;

	////KE011
	Pdc_X20DOF322_008.DOutput[1] := gInksOutputs[1].xOutPowPrintHead;
	Pdc_X20DOF322_008.DOutput[2] := gInksOutputs[2].xOutPowPrintHead;
	Pdc_X20DOF322_008.DOutput[3] := gInksOutputs[3].xOutPowPrintHead;
	Pdc_X20DOF322_008.DOutput[4] := gInksOutputs[4].xOutPowPrintHead;
	Pdc_X20DOF322_008.DOutput[5] := gInksOutputs[5].xOutPowPrintHead;
	Pdc_X20DOF322_008.DOutput[6] := gBlock[1].parSw.xEnableToPrint AND gMachine.In.xPowerSwitch;
	Pdc_X20DOF322_008.DOutput[7] := gInksOutputs[1].xOutBarResistance;
	Pdc_X20DOF322_008.DOutput[8] := gInksOutputs[2].xOutBarResistance;
	Pdc_X20DOF322_008.DOutput[9] := gInksOutputs[3].xOutBarResistance;
	Pdc_X20DOF322_008.DOutput[10] := gInksOutputs[4].xOutBarResistance;
	Pdc_X20DOF322_008.DOutput[11] := gInksOutputs[5].xOutBarResistance;
	Pdc_X20DOF322_008.DOutput[12] := gBlock[1].parSw.xEnableToPrint AND gMachine.In.xPowerSwitch;
	Pdc_X20DOF322_008.DOutput[13] := gMachine.In.xPowerSwitch;
	Pdc_X20DOF322_008.DOutput[14] := gChiller[gCuringLed[iIndexColorCuringLedBar].Parameters.iChillerIndex].Out.xStart; //gChiller[gCuringLed[iIndexColorCuringLedBar].Parameters.iChillerIndex].Out.xStart; //gCuringLed[iIndexColorCuringLedBar].Signals.Outputs.xRunChiller;
	Pdc_X20DOF322_008.DOutput[15] := gCuringLed[iIndexColorCuringLedBar].Signals.Outputs.xPowerOnLamps AND gBlockInputs[1].Safety.xSafetyOK AND gMachine.In.xPowerSwitch;
	//Pdc_X20DOF322_008.DOutput[16] := ;

	// Pdc_X20AI2636_050 THICKNESS SENSOR RESET
	Pdc_X20AI2636_050.DOutput[1] := gDing.Out.xReset;;  // Reset the target fault

	//////////
	//PRINTER
	//////////

	//gMachine.Out.xBuzzerButtonPanel ¿Donde está cableado?
	//109
//	X20DOF322_108.DOutput[1] := ;
	X20DOF322_108.DOutput[2] := gMachine.Out.xResetCB1;
	X20DOF322_108.DOutput[3] := gThicknessCtrl.Outputs.xEnableMediaSignalToCb;
	X20DOF322_108.DOutput[4] := gMachine.Out.xAirSupply;
	X20DOF322_108.DOutput[5] := gMachine.Out.xLightReset OR (gThicknessCtrl.status.MediaPosition.xMediaBelowMachine AND NOT gBelt.states.xRuningBelt AND gPLC.xBlk_100ms);

	//109
	X20DOF322_109.DOutput[1] := gJamDetect[1].Outputs.xJamTestSignal[1] OR
								gJamDetect[2].Outputs.xJamTestSignal[1];
	X20DOF322_109.DOutput[2] := gJamDetect[1].Outputs.xJamTestSignal[2] OR
								gJamDetect[2].Outputs.xJamTestSignal[2];
	X20DOF322_109.DOutput[3] := gJamDetect[1].Outputs.xJamTestSignal[3] OR
								gJamDetect[2].Outputs.xJamTestSignal[3];
	X20DOF322_109.DOutput[4] := gJamDetect[1].Outputs.xJamTestSignal[4];

	X20DOF322_109.DOutput[5] := gMachine.Out.xRemoteTeachL1;
	X20DOF322_109.DOutput[6] := gCuringLed[iIndexColorCuringLedBar].Lamp[1].Outputs.EnableLamp;
	X20DOF322_109.DOutput[7] := gCuringLed[iIndexColorCuringLedBar].Lamp[2].Outputs.EnableLamp;
	X20DOF322_109.DOutput[8] := gCuringLed[iIndexColorCuringLedBar].Lamp[3].Outputs.EnableLamp;

	//Analog outputs
	//115
	X20AO4622_115.AOutput[1] := gInksOutputs[1].iDutyCycleNegative;
	X20AO4622_115.AOutput[2] := gInksOutputs[2].iDutyCycleNegative;
	X20AO4622_115.AOutput[3] := gInksOutputs[1].iDutyCycleFilling;
	X20AO4622_115.AOutput[4] := gInksOutputs[2].iDutyCycleFilling;

	//116
	X20AO4622_116.AOutput[1] := gInksOutputs[3].iDutyCycleNegative;
	X20AO4622_116.AOutput[2] := gInksOutputs[4].iDutyCycleNegative;
	X20AO4622_116.AOutput[3] := gInksOutputs[3].iDutyCycleFilling;
	X20AO4622_116.AOutput[4] := gInksOutputs[4].iDutyCycleFilling;

	//117
	X20AO4622_117.AOutput[1] := gInksOutputs[5].iDutyCycleNegative;
	//X20AO4622_117.AOutput[2] := ;
	X20AO4622_117.AOutput[3] := gInksOutputs[5].iDutyCycleFilling;
	//X20AO4622_117.AOutput[4] := ;

	//118
	X20AO4622_118.AOutput[1] := gCuringLed[iIndexColorCuringLedBar].Lamp[1].Outputs.IntensityLampRaw;
	X20AO4622_118.AOutput[2] := gCuringLed[iIndexColorCuringLedBar].Lamp[2].Outputs.IntensityLampRaw;
	X20AO4622_118.AOutput[3] := gCuringLed[iIndexColorCuringLedBar].Lamp[3].Outputs.IntensityLampRaw;
	//X20AO4622_118.AOutput[4] := ;

	// SI UNIT BK1
	SiUnitPwrLnkBK1.Output01_16.0 := 	gBlockOutputs[1].xTrayOut; //1A
	SiUnitPwrLnkBK1.Output01_16.1 := 	gBlockOutputs[1].xTrayIn; //1B
	SiUnitPwrLnkBK1.Output01_16.2 := 	gCuringLed[iIndexColorCuringLedBar].Signals.Outputs.xPowerOnNitrogen;  //2A //[RGP] This EV has different purposes in UV and Water
	SiUnitPwrLnkBK1.Output01_16.3 := 	gBlockOutputs[1].xVenturi; //2B
	SiUnitPwrLnkBK1.Output01_16.4 := 	gTransVacuum[1].Outputs.xActiveEvToEvacuateInk; //3A
	SiUnitPwrLnkBK1.Output01_16.5 := 	gBlockOutputs[1].xWastedInkTankPump;  //4A
	SiUnitPwrLnkBK1.Output01_16.6 := 	FALSE; //5A
	SiUnitPwrLnkBK1.Output01_16.7 := 	gBlockOutputs[1].xWastedInkTankPump; //6A

	//Vacuum
//	SiUnitPwrLnkBK1.Output01_16.8 := gTransVacuum[1].Outputs.VacuumValves.0;
//	SiUnitPwrLnkBK1.Output01_16.9 := gTransVacuum[1].Outputs.VacuumValves.1;
//	SiUnitPwrLnkBK1.Output01_16.10 := gTransVacuum[1].Outputs.VacuumValves.2;
//	SiUnitPwrLnkBK1.Output01_16.11 := gTransVacuum[1].Outputs.VacuumValves.3;
//	SiUnitPwrLnkBK1.Output01_16.12 := gTransVacuum[1].Outputs.VacuumValves.4;
//	SiUnitPwrLnkBK1.Output01_16.13 := gTransVacuum[1].Outputs.VacuumValves.5;
//	SiUnitPwrLnkBK1.Output01_16.14 := gTransVacuum[1].Outputs.VacuumValves.6;
//	SiUnitPwrLnkBK1.Output01_16.15 := gTransVacuum[1].Outputs.VacuumValves.7;
//	SiUnitPwrLnkBK1.Output17_32.0 := gTransVacuum[1].Outputs.VacuumValves.8;
//	SiUnitPwrLnkBK1.Output17_32.1 := gTransVacuum[1].Outputs.VacuumValves.9;
//	SiUnitPwrLnkBK1.Output17_32.2 := gTransVacuum[1].Outputs.VacuumValves.10;
//	SiUnitPwrLnkBK1.Output17_32.3 := gTransVacuum[1].Outputs.VacuumValves.11;
//	SiUnitPwrLnkBK1.Output17_32.4 := gTransVacuum[1].Outputs.VacuumValves.12;
//	SiUnitPwrLnkBK1.Output17_32.5 := gTransVacuum[1].Outputs.VacuumValves.13;
//	SiUnitPwrLnkBK1.Output17_32.6 := gTransVacuum[1].Outputs.VacuumValves.14;
//	SiUnitPwrLnkBK1.Output17_32.7 := gTransVacuum[1].Outputs.VacuumValves.15;
//	SiUnitPwrLnkBK1.Output17_32.8 := gTransVacuum[1].Outputs.VacuumValves.16;
//	SiUnitPwrLnkBK1.Output17_32.9 := gTransVacuum[1].Outputs.VacuumValves.17;
//	SiUnitPwrLnkBK1.Output17_32.10 := gTransVacuum[1].Outputs.VacuumValves.18;
//	SiUnitPwrLnkBK1.Output17_32.11 := gTransVacuum[1].Outputs.VacuumValves.19;

	SiUnitPwrLnkBK1.Output01_16.8 := FALSE;
	SiUnitPwrLnkBK1.Output01_16.9 := FALSE;
	SiUnitPwrLnkBK1.Output01_16.10 := FALSE;
	SiUnitPwrLnkBK1.Output01_16.11 := FALSE;
	SiUnitPwrLnkBK1.Output01_16.12 := FALSE;

	SiUnitPwrLnkBK1.Output01_16.13 := gTransVacuum[1].Outputs.VacuumValves.0;
	SiUnitPwrLnkBK1.Output01_16.14 := gTransVacuum[1].Outputs.VacuumValves.1;
	SiUnitPwrLnkBK1.Output01_16.15 := gTransVacuum[1].Outputs.VacuumValves.2;
	SiUnitPwrLnkBK1.Output17_32.0 := gTransVacuum[1].Outputs.VacuumValves.3;
	SiUnitPwrLnkBK1.Output17_32.1 := gTransVacuum[1].Outputs.VacuumValves.4;
	SiUnitPwrLnkBK1.Output17_32.2 := gTransVacuum[1].Outputs.VacuumValves.5;
	SiUnitPwrLnkBK1.Output17_32.3 := gTransVacuum[1].Outputs.VacuumValves.6;
	SiUnitPwrLnkBK1.Output17_32.4 := gTransVacuum[1].Outputs.VacuumValves.7;
	SiUnitPwrLnkBK1.Output17_32.5 := gTransVacuum[1].Outputs.VacuumValves.8;
	SiUnitPwrLnkBK1.Output17_32.6 := gTransVacuum[1].Outputs.VacuumValves.9;
	SiUnitPwrLnkBK1.Output17_32.7 := gTransVacuum[1].Outputs.VacuumValves.10;
	SiUnitPwrLnkBK1.Output17_32.8 := gTransVacuum[1].Outputs.VacuumValves.11;
	SiUnitPwrLnkBK1.Output17_32.9 := gTransVacuum[1].Outputs.VacuumValves.12;
	SiUnitPwrLnkBK1.Output17_32.10 := gTransVacuum[1].Outputs.VacuumValves.13;
	SiUnitPwrLnkBK1.Output17_32.11 := gTransVacuum[1].Outputs.VacuumValves.14;
END_ACTION
```

#### OutputsMecano.st - PhysicalOutputs
```iecst
ACTION OutputsMecano:

	//////////
	//PRINTER
	//////////
	X20DOF322_108.DOutput[1] := gLine.Outputs.xGreenLight;
	X20DOF322_108.DOutput[2] := gLine.Outputs.xLightReset;
	X20DOF322_108.DOutput[3] := gLine.Outputs.xSound OR gMachine.Out.xBuzzerButtonPanel;
	X20DOF322_108.DOutput[4] := gMachine.Out.xAirSupply;
	X20DOF322_108.DOutput[5] := gLine.Outputs.xSound OR gMachine.Out.xBuzzerButtonPanel;
	X20DOF322_108.DOutput[6] := gLine.Outputs.xYellowLight;
	X20DOF322_108.DOutput[7] := gLine.Outputs.xBlueLight;
	X20DOF322_108.DOutput[8] := gLine.Outputs.xRedLight;
	X20DOF322_108.DOutput[9] := gLine.Outputs.xWhiteLight;
	//X20DOF322_108.DOutput[10] := ;
	X20DOF322_108.DOutput[11] := gJamDetect[1].Outputs.xJamTestSignal[1] OR
								gJamDetect[2].Outputs.xJamTestSignal[1] OR
								gJamDetect[3].Outputs.xJamTestSignal[1];
	X20DOF322_108.DOutput[12] := gJamDetect[1].Outputs.xJamTestSignal[2] OR
								gJamDetect[2].Outputs.xJamTestSignal[2] OR
								gJamDetect[3].Outputs.xJamTestSignal[2];
	X20DOF322_108.DOutput[13] := gJamDetect[1].Outputs.xJamTestSignal[3] OR
								gJamDetect[2].Outputs.xJamTestSignal[3] OR
								gJamDetect[3].Outputs.xJamTestSignal[3];
	X20DOF322_108.DOutput[14] := gJamDetect[1].Outputs.xJamTestSignal[4] OR
								gJamDetect[2].Outputs.xJamTestSignal[4] OR
								gJamDetect[3].Outputs.xJamTestSignal[4];

	X20DOF322_109.DOutput[1] := gMachine.Out.xRemoteTeachL1;
	X20DOF322_109.DOutput[2] := gMachine.Out.xRemoteTeachL2;
	X20DOF322_109.DOutput[3] := gThicknessCtrl.Outputs.xEnableMediaSignalToCb;
	//X20DOF322_109.DOutput[4] := ;
	X20DOF322_109.DOutput[5] := gMachine.Out.xResetCB1 OR gMachine.Out.xResetCB2;
	X20DOF322_109.DOutput[6] := gMachine.Out.xResetRouter;

	X20DOF322_110.DOutput[1] := gInksOutputs[3].xOutPowPrintHead;
	X20DOF322_110.DOutput[2] := gInksOutputs[4].xOutPowPrintHead;
	X20DOF322_110.DOutput[3] := gInksOutputs[5].xOutPowPrintHead;
	X20DOF322_110.DOutput[4] := gInksOutputs[6].xOutPowPrintHead;
	X20DOF322_110.DOutput[5] := gInksOutputs[7].xOutPowPrintHead;
	X20DOF322_110.DOutput[6] := gInksOutputs[8].xOutPowPrintHead;
	X20DOF322_110.DOutput[7] := gInksOutputs[9].xOutPowPrintHead;
	X20DOF322_110.DOutput[8] := gInksOutputs[10].xOutPowPrintHead;
	X20DOF322_110.DOutput[9] := gInksOutputs[3].xOutBarResistance;
	X20DOF322_110.DOutput[10] := gInksOutputs[4].xOutBarResistance;
	X20DOF322_110.DOutput[11] := gInksOutputs[5].xOutBarResistance;
	X20DOF322_110.DOutput[12] := gInksOutputs[6].xOutBarResistance;
	X20DOF322_110.DOutput[13] := gInksOutputs[7].xOutBarResistance;
	X20DOF322_110.DOutput[14] := gInksOutputs[8].xOutBarResistance;
	X20DOF322_110.DOutput[15] := gInksOutputs[9].xOutBarResistance;
	X20DOF322_110.DOutput[16] := gInksOutputs[10].xOutBarResistance;

	//Analog outputs
	X20AO4622_116.AOutput[1] := gInksOutputs[3].iDutyCycleFilling;
	X20AO4622_116.AOutput[2] := gInksOutputs[4].iDutyCycleFilling;
 	X20AO4622_116.AOutput[3] := gInksOutputs[3].iDutyCycleNegative;
	X20AO4622_116.AOutput[4] := gInksOutputs[4].iDutyCycleNegative;
 	X20AO4622_117.AOutput[1] := gInksOutputs[5].iDutyCycleFilling;
	X20AO4622_117.AOutput[2] := gInksOutputs[6].iDutyCycleFilling;
 	X20AO4622_117.AOutput[3] := gInksOutputs[5].iDutyCycleNegative;
	X20AO4622_117.AOutput[4] := gInksOutputs[6].iDutyCycleNegative;
	X20AO4622_118.AOutput[1] := gInksOutputs[7].iDutyCycleFilling;
	X20AO4622_118.AOutput[2] := gInksOutputs[8].iDutyCycleFilling;
	X20AO4622_118.AOutput[3] := gInksOutputs[7].iDutyCycleNegative;
	X20AO4622_118.AOutput[4] := gInksOutputs[8].iDutyCycleNegative;
	X20AO4622_119.AOutput[1] := gInksOutputs[9].iDutyCycleFilling;
	X20AO4622_119.AOutput[2] := gInksOutputs[10].iDutyCycleFilling;
	X20AO4622_119.AOutput[3] := gInksOutputs[9].iDutyCycleNegative;
	X20AO4622_119.AOutput[4] := gInksOutputs[10].iDutyCycleNegative;

	X20DOF322_155.DOutput[1] := gCuringLed[iIndexColorCuringLedBar].Lamp[1].Outputs.EnableLamp;
	X20DOF322_155.DOutput[2] := gCuringLed[iIndexColorCuringLedBar].Lamp[2].Outputs.EnableLamp;
	X20DOF322_155.DOutput[3] := gCuringLed[iIndexColorCuringLedBar].Lamp[3].Outputs.EnableLamp;
	X20DOF322_155.DOutput[4] := gCuringLed[iIndexColorCuringLedBar].Lamp[4].Outputs.EnableLamp;
	X20DOF322_155.DOutput[5] := gCuringLed[iIndexColorCuringLedBar].Lamp[5].Outputs.EnableLamp;
	//X20DOF322_155.DOutput[6] := ;
	X20DOF322_155.DOutput[7] := gCuringLed[iIndexWhiteCuringLedBar].Lamp[1].Outputs.EnableLamp;
	X20DOF322_155.DOutput[8] := gCuringLed[iIndexWhiteCuringLedBar].Lamp[2].Outputs.EnableLamp;
	X20DOF322_155.DOutput[9] := gCuringLed[iIndexWhiteCuringLedBar].Lamp[3].Outputs.EnableLamp;
	X20DOF322_155.DOutput[10] := gCuringLed[iIndexWhiteCuringLedBar].Lamp[4].Outputs.EnableLamp;
	X20DOF322_155.DOutput[11] := gCuringLed[iIndexWhiteCuringLedBar].Lamp[5].Outputs.EnableLamp;

	X20DOF322_156.DOutput[1] := gCuringLed[iIndexPrimerCuringLedBar].Lamp[1].Outputs.EnableLamp;
	X20DOF322_156.DOutput[2] := gCuringLed[iIndexPrimerCuringLedBar].Lamp[2].Outputs.EnableLamp;
	X20DOF322_156.DOutput[3] := gCuringLed[iIndexPrimerCuringLedBar].Lamp[3].Outputs.EnableLamp;
	X20DOF322_156.DOutput[4] := gCuringLed[iIndexPrimerCuringLedBar].Lamp[4].Outputs.EnableLamp;
	X20DOF322_156.DOutput[5] := gCuringLed[iIndexPrimerCuringLedBar].Lamp[5].Outputs.EnableLamp;

	X20DOF322_156.DOutput[12] := gMachine.Out.xAntiStaticPOn;
	X20DOF322_156.DOutput[13] := gMachine.commands.CleanBelt.xCleanBeltMoveFwd;
	X20DOF322_156.DOutput[14] := gMachine.commands.CleanBelt.xCleanBeltMoveBwd;
	X20DOF322_156.DOutput[15] := gMachine.commands.CleanBelt.xCleanBeltResetRelay;

	//Analog outputs
	X20AO4622_158.AOutput[1] := gCuringLed[iIndexColorCuringLedBar].Lamp[1].Outputs.IntensityLampRaw;
	X20AO4622_158.AOutput[2] := gCuringLed[iIndexColorCuringLedBar].Lamp[2].Outputs.IntensityLampRaw;
	X20AO4622_158.AOutput[3] := gCuringLed[iIndexColorCuringLedBar].Lamp[3].Outputs.IntensityLampRaw;
	X20AO4622_158.AOutput[4] := gCuringLed[iIndexColorCuringLedBar].Lamp[4].Outputs.IntensityLampRaw;

	X20AO4622_159.AOutput[1] := gCuringLed[iIndexColorCuringLedBar].Lamp[5].Outputs.IntensityLampRaw;
	//X20AO4622_159.AOutput[2] := ;
	X20AO4622_159.AOutput[3] := gCuringLed[iIndexWhiteCuringLedBar].Lamp[1].Outputs.IntensityLampRaw;
	X20AO4622_159.AOutput[4] := gCuringLed[iIndexWhiteCuringLedBar].Lamp[2].Outputs.IntensityLampRaw;

	X20AO4622_160.AOutput[1] := gCuringLed[iIndexWhiteCuringLedBar].Lamp[3].Outputs.IntensityLampRaw;
	X20AO4622_160.AOutput[2] := gCuringLed[iIndexWhiteCuringLedBar].Lamp[4].Outputs.IntensityLampRaw;
	X20AO4622_160.AOutput[3] := gCuringLed[iIndexWhiteCuringLedBar].Lamp[5].Outputs.IntensityLampRaw;
	X20AO4622_160.AOutput[4] := gCuringLed[iIndexPrimerCuringLedBar].Lamp[1].Outputs.IntensityLampRaw;

	X20AO4622_161.AOutput[1] := gCuringLed[iIndexPrimerCuringLedBar].Lamp[2].Outputs.IntensityLampRaw;
	X20AO4622_161.AOutput[2] := gCuringLed[iIndexPrimerCuringLedBar].Lamp[3].Outputs.IntensityLampRaw;
	X20AO4622_161.AOutput[3] := gCuringLed[iIndexPrimerCuringLedBar].Lamp[4].Outputs.IntensityLampRaw;
	X20AO4622_161.AOutput[4] := gCuringLed[iIndexPrimerCuringLedBar].Lamp[5].Outputs.IntensityLampRaw;

	//////////
	//PDC
	//////////
	Pdc_X20DOF322_009.DOutput[1] := gMachine.In.xPowerSwitch;
	Pdc_X20DOF322_009.DOutput[2] := gLine.Outputs.ExternalDevices[10].xClose; //Primer
	Pdc_X20DOF322_009.DOutput[3] := gLine.Outputs.ExternalDevices[10].xOpen;
	Pdc_X20DOF322_009.DOutput[4] := gOverVarnish.Outputs.Physical.xRunDryer;
	Pdc_X20DOF322_009.DOutput[5] := gOverVarnish.Outputs.Physical.xRunTransport;
	Pdc_X20DOF322_009.DOutput[6] := gOverVarnish.Outputs.Physical.xRunPriming;
	Pdc_X20DOF322_009.DOutput[7] := gOverVarnish.Outputs.Physical.xPrepareToPrime;
	//Pdc_X20DOF322_009.DOutput[8] := ;
	//Pdc_X20DOF322_009.DOutput[9] := ;
	Pdc_X20DOF322_009.DOutput[10] := gLine.Outputs.ExternalDevices[1].xClose; //Opv
	Pdc_X20DOF322_009.DOutput[11] := gLine.Outputs.ExternalDevices[1].xOpen;
	Pdc_X20DOF322_009.DOutput[12] := gPrimer.Outputs.Physical.xRunDryer;
	Pdc_X20DOF322_009.DOutput[13] := gPrimer.Outputs.Physical.xRunTransport;
	Pdc_X20DOF322_009.DOutput[14] := gPrimer.Outputs.Physical.xRunPriming;
	Pdc_X20DOF322_009.DOutput[15] := gPrimer.Outputs.Physical.xPrepareToPrime;
	//Pdc_X20DOF322_009.DOutput[16] := ;

	//Pdc_X20DOF322_010
	Pdc_X20DOF322_010.DOutput[1] := gLine.Outputs.ExternalDevices[0].xClose; //Feeder
	Pdc_X20DOF322_010.DOutput[2] := gFeeder.Outputs.Physical.xPrepareToFeed;
	Pdc_X20DOF322_010.DOutput[3] := gFeeder.Outputs.Physical.xStartFeeding;
	Pdc_X20DOF322_010.DOutput[4] := gFeeder.Outputs.Physical.xFastStop;
	Pdc_X20DOF322_010.DOutput[5] := gLine.Outputs.ExternalDevices[11].xClose; //Sarm
	Pdc_X20DOF322_010.DOutput[6] := gSarm.Outputs.xStartTransport;
	Pdc_X20DOF322_010.DOutput[7] := gSarm.Outputs.xFastStop;
	Pdc_X20DOF322_010.DOutput[8] := gLine.Outputs.ExternalDevices[6].xClose; //Stacker
	Pdc_X20DOF322_010.DOutput[9] := gStacker.Outputs.xRun;
	Pdc_X20DOF322_010.DOutput[10] := gThicknessCtrl.Outputs.xReject; //gStacker.Outputs.xRejectSheet;
	Pdc_X20DOF322_010.DOutput[11] := gStacker.Outputs.xPrepareToStack;
	Pdc_X20DOF322_010.DOutput[12] := gStacker.Outputs.xEjectRejectStack;
	Pdc_X20DOF322_010.DOutput[13] := gStacker.Outputs.xStackEject;
	Pdc_X20DOF322_010.DOutput[14] := FALSE;
	Pdc_X20DOF322_010.DOutput[15] := FALSE;
	Pdc_X20DOF322_010.DOutput[16] := FALSE;

	Pdc_X20DOF322_011.DOutput[1] := gMachine.Out.xResetHub;
	Pdc_X20DOF322_011.DOutput[2] := gMachine.Out.xResetSwitch;
	Pdc_X20DOF322_011.DOutput[3] := gMachine.Out.xResetSwitch;
	Pdc_X20DOF322_011.DOutput[4] := gMachine.Out.xSuctionTurbine;
//	Pdc_X20DOF322_011.DOutput[5] := ;
//	Pdc_X20DOF322_011.DOutput[6] := ;
//	Pdc_X20DOF322_011.DOutput[7] := ;

	//Line X20DOF322_023
	Pdc_X20DOF322_025.DOutput[1] := gChiller[1].St.xInstalled;
	Pdc_X20DOF322_025.DOutput[2] := gChiller[1].Out.xStart;
	Pdc_X20DOF322_025.DOutput[3] := gChiller[2].St.xInstalled;
	Pdc_X20DOF322_025.DOutput[4] := gChiller[2].Out.xStart;
//	Pdc_X20DOF322_025.DOutput[5] := NOT gSafetyController.Alarms.xAlrPrinter;
//	Pdc_X20DOF322_025.DOutput[6] := gChiller[3].Out.xStart;
//	Pdc_X20DOF322_025.DOutput[7] := Chiller de printheads?;
//	Pdc_X20DOF322_025.DOutput[8] := Chiller de printheads?;
	Pdc_X20DOF322_025.DOutput[9] := NOT (gLine.Outputs.ExternalDevices[7].xClose AND gCuringLed[iIndexColorCuringLedBar].Signals.Outputs.xPowerOnLamps AND NOT gSafetyController.Alarms.xAlrPrinter AND gLine.Inputs.xPrinterPowered); //96VDC Powersupplies inhibit signal
	Pdc_X20DOF322_025.DOutput[10] := NOT (gLine.Outputs.ExternalDevices[7].xClose AND gCuringLed[iIndexWhiteCuringLedBar].Signals.Outputs.xPowerOnLamps AND NOT gSafetyController.Alarms.xAlrPrinter AND gLine.Inputs.xPrinterPowered); //96VDC Powersupplies inhibit signal
	Pdc_X20DOF322_025.DOutput[11] := NOT (gLine.Outputs.ExternalDevices[7].xClose AND gCuringLed[iIndexPrimerCuringLedBar].Signals.Outputs.xPowerOnLamps AND NOT gSafetyController.Alarms.xAlrPrinter AND gLine.Inputs.xPrinterPowered); //96VDC Powersupplies inhibit signal

	// SI UNIT BK1 PNEUMATIC DIAGRAM V03
	SiUnitPwrLnkBK1.Output01_16.0 := 	gBlockOutputs[1].xTrayIn; //1A
	SiUnitPwrLnkBK1.Output01_16.1 := 	gBlockOutputs[1].xTrayOut; //1B
	SiUnitPwrLnkBK1.Output01_16.2 := 	gMachine.commands.CleanBelt.xCleanBeltPump OR
										gCuringLed[iIndexWhiteCuringLedBar].Signals.Outputs.xPowerOnNitrogen OR
										gCuringLed[iIndexColorCuringLedBar].Signals.Outputs.xPowerOnNitrogen OR
										gCuringLed[iIndexPrimerCuringLedBar].Signals.Outputs.xPowerOnNitrogen; //2A //[RGP] This EV has different purposes in UV and Water
	SiUnitPwrLnkBK1.Output01_16.3 := 	gBlockOutputs[1].xVenturi; //2B
	SiUnitPwrLnkBK1.Output01_16.4 := 	gBlockOutputs[1].xCleaningWaterPump; //3A
	SiUnitPwrLnkBK1.Output01_16.5 := 	gMachine.commands.CleanBelt.xPistonFlojet;  //4A
	SiUnitPwrLnkBK1.Output01_16.6 := 	FALSE; //5A
	SiUnitPwrLnkBK1.Output01_16.7 := 	gBlockOutputs[1].xCappingWaterPump OR gBlockOutputs[1].xWastedInkTankPump; //6A

	//Vacuum
	SiUnitPwrLnkBK1.Output01_16.10 := gTransVacuum[1].Outputs.VacuumValves.0; //8A
	SiUnitPwrLnkBK1.Output01_16.11 := gTransVacuum[1].Outputs.VacuumValves.1; //8B
	SiUnitPwrLnkBK1.Output01_16.12 := gTransVacuum[1].Outputs.VacuumValves.2; //9A
	SiUnitPwrLnkBK1.Output01_16.13 := gTransVacuum[1].Outputs.VacuumValves.3; //9B
	SiUnitPwrLnkBK1.Output01_16.14 := gTransVacuum[1].Outputs.VacuumValves.4; //10A
	SiUnitPwrLnkBK1.Output01_16.15 := gTransVacuum[1].Outputs.VacuumValves.5; //10B
	SiUnitPwrLnkBK1.Output17_32.0 := gTransVacuum[1].Outputs.VacuumValves.6; //11A
	SiUnitPwrLnkBK1.Output17_32.1 := gTransVacuum[1].Outputs.VacuumValves.7; //11B
	SiUnitPwrLnkBK1.Output17_32.2 := gTransVacuum[1].Outputs.VacuumValves.8; //12A
	SiUnitPwrLnkBK1.Output17_32.3 := gTransVacuum[1].Outputs.VacuumValves.9; //12B
	SiUnitPwrLnkBK1.Output17_32.4 := gTransVacuum[1].Outputs.VacuumValves.10; //13A
	SiUnitPwrLnkBK1.Output17_32.5 := gTransVacuum[1].Outputs.VacuumValves.11; //13B
	SiUnitPwrLnkBK1.Output17_32.6 := gTransVacuum[1].Outputs.VacuumValves.12; //14A
	SiUnitPwrLnkBK1.Output17_32.7 := gTransVacuum[1].Outputs.VacuumValves.13; //14B
	SiUnitPwrLnkBK1.Output17_32.8 := gTransVacuum[1].Outputs.VacuumValves.14; //15A
	SiUnitPwrLnkBK1.Output17_32.9 := gTransVacuum[1].Outputs.VacuumValves.15; //15B
	SiUnitPwrLnkBK1.Output17_32.10 := gTransVacuum[1].Outputs.VacuumValves.16; //16A
	SiUnitPwrLnkBK1.Output17_32.11 := gTransVacuum[1].Outputs.VacuumValves.17; //16B

END_ACTION
```

### Package Logical/Printer/BlockSignalsManager - Logical to Physical map

### Program Logical/Printer/BlockSignalsManager/BlockInputsMapping (IEC) - Input logical

#### BlockInputsMapping.st - Init, cyclic, exit code
```iecst
PROGRAM _CYCLIC

		//If in automation runtime, do not assign physical mapping
	IF gMachine.St.HwData.Family = FAMILY_BRAUTOMATIONRUNTIME THEN
		RETURN;
	END_IF

	FOR iIndexBlockIn := GC_FIRST_BLOCK TO gMachine.Pt.CT.iNumBlocks DO
		// gBlockOutputs is stBlock_Inputs
		gBlock[iIndexBlockIn].In := gBlockInputs[gBlock[iIndexBlockIn].parameters.iMappingBlock];

	END_FOR;

	//////////////////////////////////////////
	// JAM INPUTS ASSIGNATION
	IF NOT gMachine.parSw.xJamDetectEnable THEN
		RETURN;
	END_IF

	FOR iIndexJam:=1 TO gMachine.St.iJamDevices DO

		//Reference working data to the general data
		dataJam ACCESS ADR(gJamDetect[iIndexJam]);

		IF dataJam.Parameters.iMappingJam > 0 AND dataJam.Parameters.iMappingJam <= MAX_LAST_JAMDEVICE THEN
			dataJam.Inputs := gJamInputs[dataJam.Parameters.iMappingJam];
		END_IF

	END_FOR;

END_PROGRAM
```

### Package Logical/Printer/InksSignals - Inputs and outputs assignation

- Program Logical/Printer/InksSignals/InksInputs (IEC) - Inputs assignation (no source held here)

### Program Logical/Printer/InksSignals/InksOutputs (IEC) - Outputs assignation

#### InksOutputs.st - Cyclic code
```iecst
PROGRAM _CYCLIC
	(* Insert code here *)

	FOR iIndexInksOut:=1 TO MAX_LAST_INK DO

		//Reference working data to the general data
		dataInksOut ACCESS ADR(gInks[iIndexInksOut]);

		IF dataInksOut.parSw.Config.iMappingBar >= 1 AND dataInksOut.parSw.Config.iMappingBar <= MAX_LAST_INK THEN
			gInksOutputs[dataInksOut.parSw.Config.iMappingBar]:= dataInksOut.signals.out;
		END_IF

	END_FOR;

	// ####################################################################
	// ####################################################################
	//  Reset bar outputs if do not have any logical bar mapped
	// ####################################################################

	// Reset the index if the index is not valid
	IF iIndexPhysicalInksSlow = 0 OR iIndexPhysicalInksSlow > MAX_LAST_INK THEN
		//Resetart index
		iIndexPhysicalInksSlow := 1;
		iIndexInksSlow := 1;
	END_IF
	IF iIndexInksSlow = 0 OR iIndexInksSlow > MAX_LAST_INK THEN iIndexInksSlow := 1; END_IF

	//If the physical bar has a logical bar in that position, go to next physical bar and reset logical index bar
	IF iIndexPhysicalInksSlow = INT_TO_USINT(gInks[iIndexInksSlow].parSw.Config.iMappingBar) THEN
		iIndexPhysicalInksSlow := iIndexPhysicalInksSlow + 1;
		iIndexInksSlow := 1;
	ELSE
		iIndexInksSlow := iIndexInksSlow + 1;
	END_IF

	//If there is no logical bar with the mapping of the physical position, reset the outputs
	IF iIndexInksSlow > MAX_LAST_INK THEN

		//Reset the outputs to avoid keeping the outputs active
		gInksOutputs[iIndexPhysicalInksSlow] := inksOutputsReseted;

		//Go to next physical and reset logical index bar
		iIndexPhysicalInksSlow := iIndexPhysicalInksSlow + 1;
		iIndexInksSlow := 1;
	END_IF

END_PROGRAM
```

#### InksOutputs.var - Local variables
```iecst
VAR
	iIndexInksOut : USINT;
	dataInksOut : REFERENCE TO stInks;
	iIndexInksSlow : USINT;
	iIndexPhysicalInksSlow : USINT;
	inksOutputsReseted : stInksSignalsOut;
END_VAR
```

### ReadmeInksInOut.txt - InksInOut package instructions
```
	(* From efi Cretaprint Almazora Castellon

	*)
```

### Package Logical/Printer/Comms - Communication PC  PLC

### Comms.var
```iecst
VAR
	FB_BRSE_MBT_Server : BRSE_MBT_Server := (0);
END_VAR
VAR RETAIN
	HoldingRegister : ARRAY[0..8999] OF INT;
END_VAR
VAR CONSTANT
	SERIAL_NAME_ASSIGNATION_ADR : UINT := 900;
	SERIAL_NAME_TRIGGER_ADR : UINT := 949;
	SERIAL_NAME_STATUS_ADR : UINT := 950;
END_VAR
```

### Program Logical/Printer/Comms/Kernel2PLC (IEC)

#### Kernel2PLC.st - Cyclic code
```iecst
PROGRAM _CYCLIC

	//If in Simulation and running without Kernel, do not execute communications
	IF gMachine.St.HwData.Family = FAMILY_BRAUTOMATIONRUNTIME AND (NOT gSimMachine.Parameters.xRunWithKernel OR gMachine.Pt.CommsType=NoCommsType)  THEN
		RETURN;
	END_IF

	IF gMachine.Pt.CommsType=Type_ModbusTcp THEN
		Kernel2PLC_AutoCode;
	END_IF

	ReadSerialName;

END_PROGRAM
```
